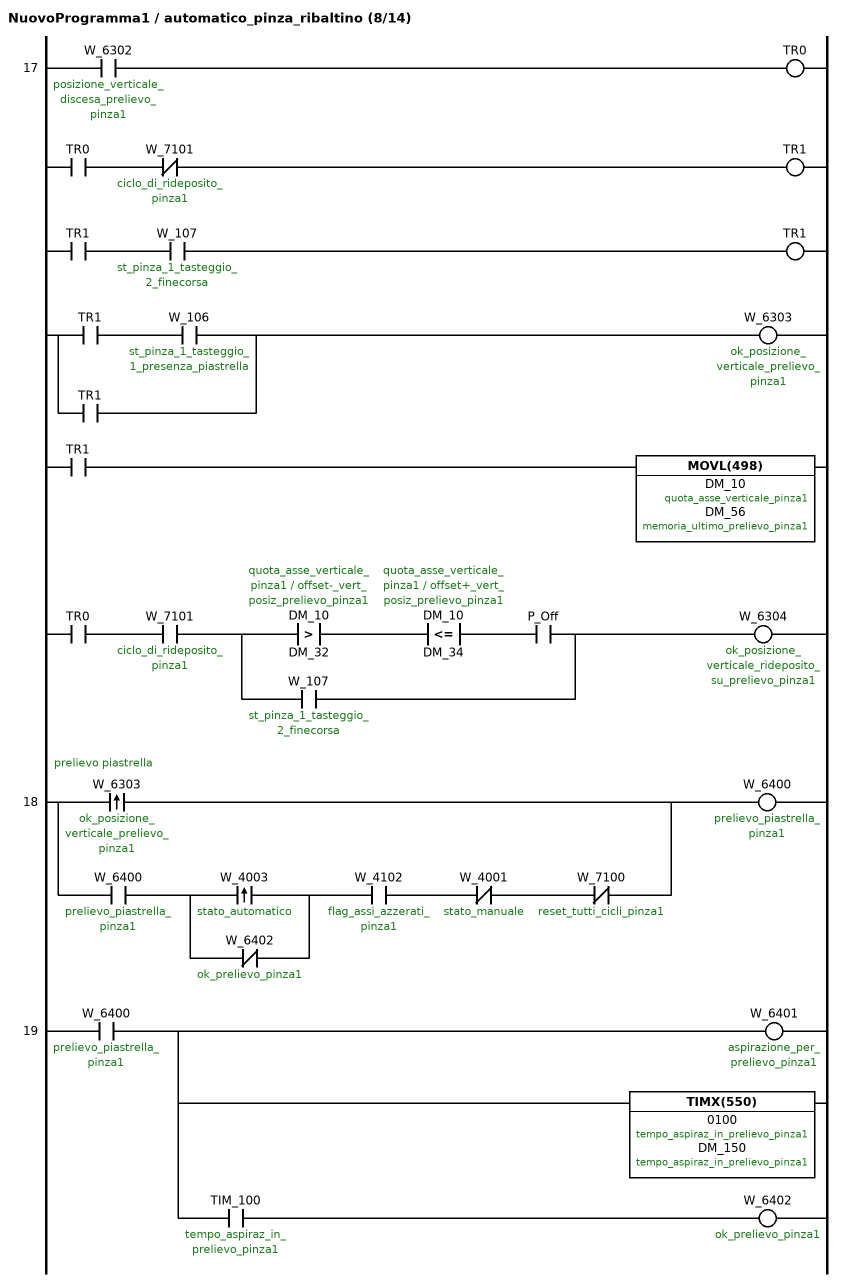
; [picture p48: NuovoProgramma1 / automatico_pinza_ribaltino, rungs 17-19]
; rung 17
LD W_6302  ; posizione_verticale_discesa_prelievo_pinza1
OUT TR0
ANDNOT W_7101  ; ciclo_di_rideposito_pinza1
OUT TR1
AND W_106  ; st_pinza_1_tasteggio_1_presenza_piastrella
LD TR1
AND W_107  ; st_pinza_1_tasteggio_2_finecorsa
OUT TR1
ORLD
OUT W_6303  ; ok_posizione_verticale_prelievo_pinza1
LD TR1
MOVL(498) DM_10 DM_56  ; quota_asse_verticale_pinza1, memoria_ultimo_prelievo_pinza1
LD TR0
AND W_7101  ; ciclo_di_rideposito_pinza1
LD>SL(323) DM_10 DM_32  ; quota_asse_verticale_pinza1, offset-_vert_posiz_prelievo_pinza1
AND<=SL(318) DM_10 DM_34  ; quota_asse_verticale_pinza1, offset+_vert_posiz_prelievo_pinza1
AND P_Off
OR W_107  ; st_pinza_1_tasteggio_2_finecorsa
ANDLD
OUT W_6304  ; ok_posizione_verticale_rideposito_su_prelievo_pinza1
; rung 18: prelievo piastrella
@LD W_6303  ; ok_posizione_verticale_prelievo_pinza1
LD W_6400  ; prelievo_piastrella_pinza1
@LD W_4003  ; stato_automatico
ORNOT W_6402  ; ok_prelievo_pinza1
ANDLD
AND W_4102  ; flag_assi_azzerati_pinza1
ANDNOT W_4001  ; stato_manuale
ANDNOT W_7100  ; reset_tutti_cicli_pinza1
ORLD
OUT W_6400  ; prelievo_piastrella_pinza1
; rung 19
LD W_6400  ; prelievo_piastrella_pinza1
OUT W_6401  ; aspirazione_per_prelievo_pinza1
TIMX(550) 0100 DM_150  ; tempo_aspiraz_in_prelievo_pinza1
AND TIM_100  ; tempo_aspiraz_in_prelievo_pinza1
OUT W_6402  ; ok_prelievo_pinza1

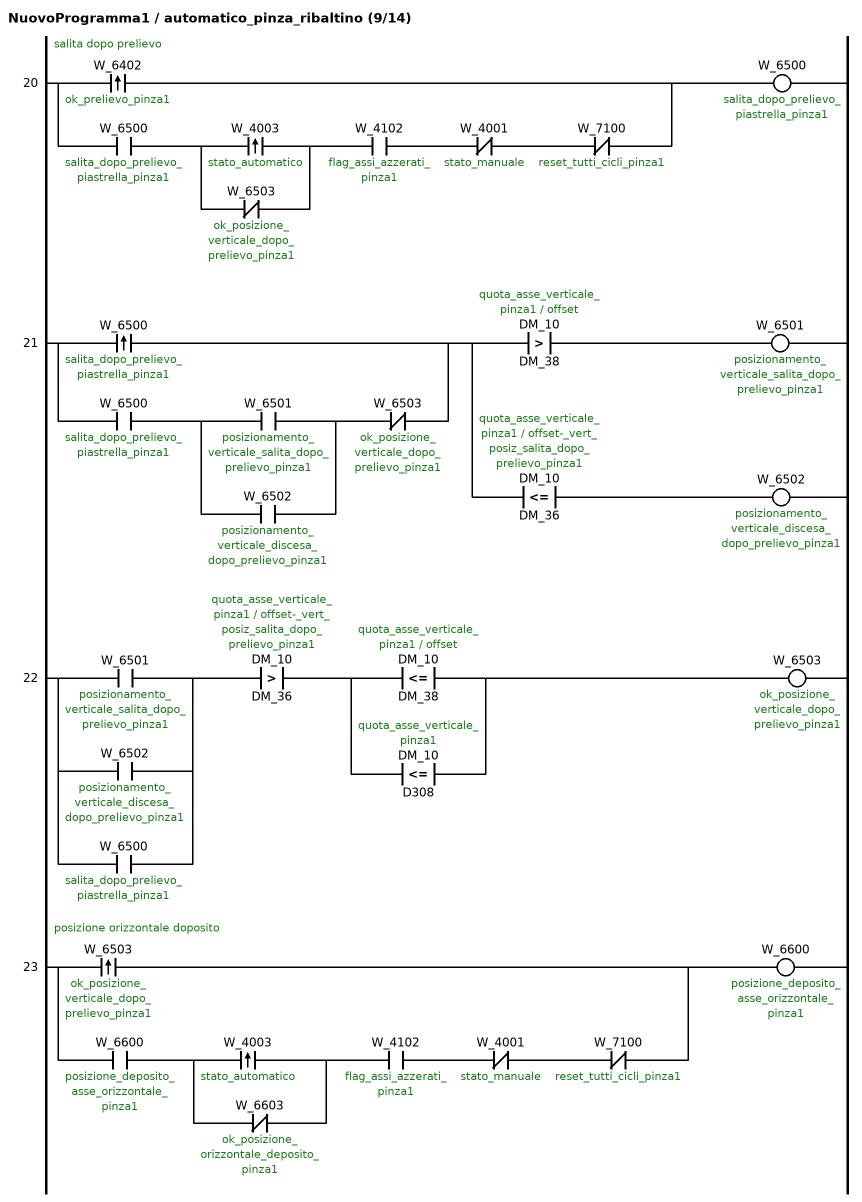
; rung 20: salita dopo prelievo
@LD W_6402  ; ok_prelievo_pinza1
LD W_6500  ; salita_dopo_prelievo_piastrella_pinza1
@LD W_4003  ; stato_automatico
ORNOT W_6503  ; ok_posizione_verticale_dopo_prelievo_pinza1
ANDLD
AND W_4102  ; flag_assi_azzerati_pinza1
ANDNOT W_4001  ; stato_manuale
ANDNOT W_7100  ; reset_tutti_cicli_pinza1
ORLD
OUT W_6500  ; salita_dopo_prelievo_piastrella_pinza1
; rung 21
@LD W_6500  ; salita_dopo_prelievo_piastrella_pinza1
LD W_6500  ; salita_dopo_prelievo_piastrella_pinza1
LD W_6501  ; posizionamento_verticale_salita_dopo_prelievo_pinza1
OR W_6502  ; posizionamento_verticale_discesa_dopo_prelievo_pinza1
ANDLD
ANDNOT W_6503  ; ok_posizione_verticale_dopo_prelievo_pinza1
ORLD
OUT TR0
AND>SL(323) DM_10 DM_38  ; quota_asse_verticale_pinza1, offset
OUT W_6501  ; posizionamento_verticale_salita_dopo_prelievo_pinza1
LD TR0
AND<=SL(318) DM_10 DM_36  ; quota_asse_verticale_pinza1, offset-_vert_posiz_salita_dopo_prelievo_pinza1
OUT W_6502  ; posizionamento_verticale_discesa_dopo_prelievo_pinza1
; rung 22
LD W_6501  ; posizionamento_verticale_salita_dopo_prelievo_pinza1
OR W_6502  ; posizionamento_verticale_discesa_dopo_prelievo_pinza1
OR W_6500  ; salita_dopo_prelievo_piastrella_pinza1
AND>SL(323) DM_10 DM_36  ; quota_asse_verticale_pinza1, offset-_vert_posiz_salita_dopo_prelievo_pinza1
LD<=SL(318) DM_10 DM_38  ; quota_asse_verticale_pinza1, offset
OR<=SL(318) DM_10 D308  ; quota_asse_verticale_pinza1
ANDLD
OUT W_6503  ; ok_posizione_verticale_dopo_prelievo_pinza1
; rung 23: posizione orizzontale doposito
@LD W_6503  ; ok_posizione_verticale_dopo_prelievo_pinza1
LD W_6600  ; posizione_deposito_asse_orizzontale_pinza1
@LD W_4003  ; stato_automatico
ORNOT W_6603  ; ok_posizione_orizzontale_deposito_pinza1
ANDLD
AND W_4102  ; flag_assi_azzerati_pinza1
ANDNOT W_4001  ; stato_manuale
ANDNOT W_7100  ; reset_tutti_cicli_pinza1
ORLD
OUT W_6600  ; posizione_deposito_asse_orizzontale_pinza1

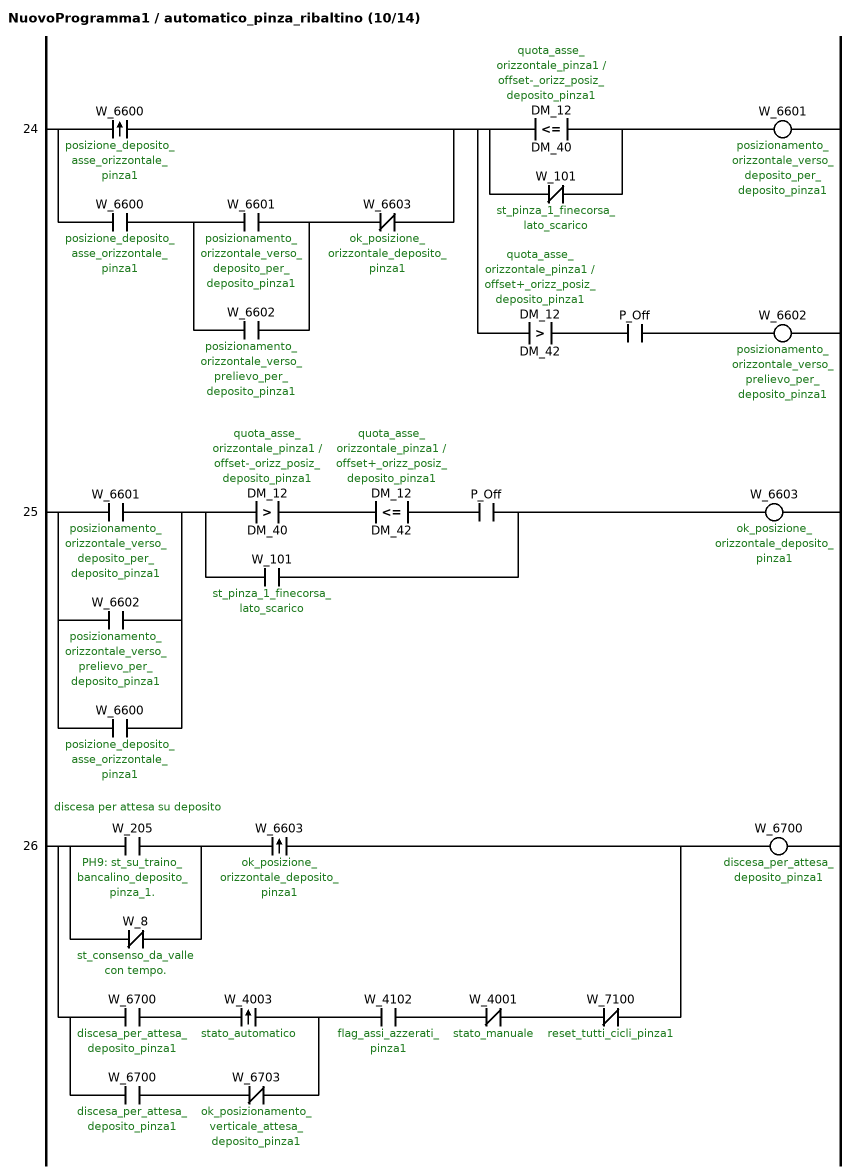
; rung 24
@LD W_6600  ; posizione_deposito_asse_orizzontale_pinza1
LD W_6600  ; posizione_deposito_asse_orizzontale_pinza1
LD W_6601  ; posizionamento_orizzontale_verso_deposito_per_deposito_pinza1
OR W_6602  ; posizionamento_orizzontale_verso_prelievo_per_deposito_pinza1
ANDLD
ANDNOT W_6603  ; ok_posizione_orizzontale_deposito_pinza1
ORLD
OUT TR0
LD<=SL(318) DM_12 DM_40  ; quota_asse_orizzontale_pinza1, offset-_orizz_posiz_deposito_pinza1
ORNOT W_101  ; st_pinza_1_finecorsa_lato_scarico
ANDLD
OUT W_6601  ; posizionamento_orizzontale_verso_deposito_per_deposito_pinza1
LD TR0
AND>SL(323) DM_12 DM_42  ; quota_asse_orizzontale_pinza1, offset+_orizz_posiz_deposito_pinza1
AND P_Off
OUT W_6602  ; posizionamento_orizzontale_verso_prelievo_per_deposito_pinza1
; rung 25
LD W_6601  ; posizionamento_orizzontale_verso_deposito_per_deposito_pinza1
OR W_6602  ; posizionamento_orizzontale_verso_prelievo_per_deposito_pinza1
OR W_6600  ; posizione_deposito_asse_orizzontale_pinza1
LD>SL(323) DM_12 DM_40  ; quota_asse_orizzontale_pinza1, offset-_orizz_posiz_deposito_pinza1
AND<=SL(318) DM_12 DM_42  ; quota_asse_orizzontale_pinza1, offset+_orizz_posiz_deposito_pinza1
AND P_Off
OR W_101  ; st_pinza_1_finecorsa_lato_scarico
ANDLD
OUT W_6603  ; ok_posizione_orizzontale_deposito_pinza1
; rung 26: discesa per attesa su deposito
LD W_205  ; PH9: st_su_traino_bancalino_deposito_pinza_1.
ORNOT W_8  ; st_consenso_da_valle con tempo.
@AND W_6603  ; ok_posizione_orizzontale_deposito_pinza1
LD W_6700  ; discesa_per_attesa_deposito_pinza1
@AND W_4003  ; stato_automatico
LD W_6700  ; discesa_per_attesa_deposito_pinza1
ANDNOT W_6703  ; ok_posizionamento_verticale_attesa_deposito_pinza1
ORLD
AND W_4102  ; flag_assi_azzerati_pinza1
ANDNOT W_4001  ; stato_manuale
ANDNOT W_7100  ; reset_tutti_cicli_pinza1
ORLD
OUT W_6700  ; discesa_per_attesa_deposito_pinza1

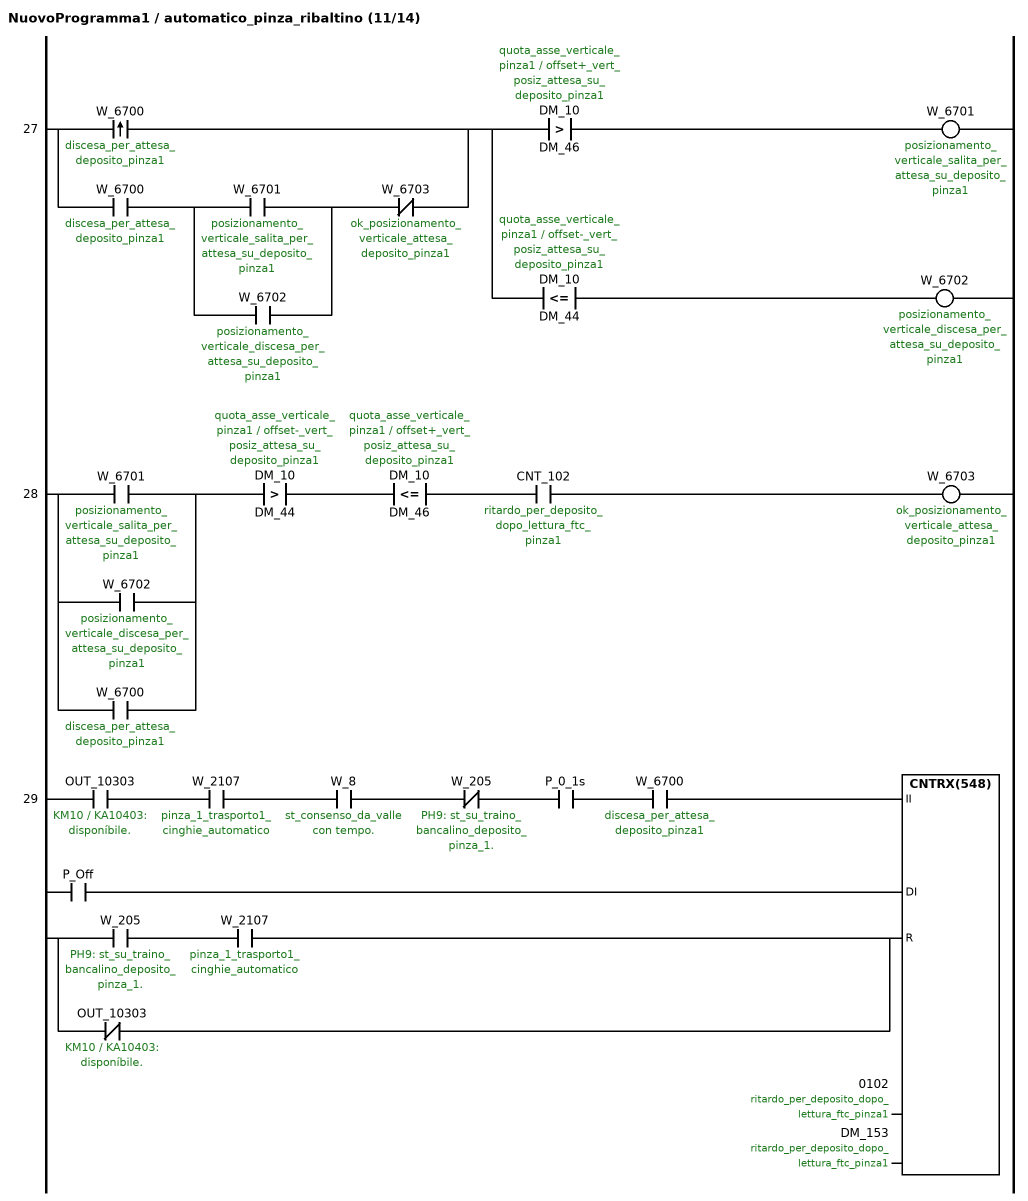
; rung 27
@LD W_6700  ; discesa_per_attesa_deposito_pinza1
LD W_6700  ; discesa_per_attesa_deposito_pinza1
LD W_6701  ; posizionamento_verticale_salita_per_attesa_su_deposito_pinza1
OR W_6702  ; posizionamento_verticale_discesa_per_attesa_su_deposito_pinza1
ANDLD
ANDNOT W_6703  ; ok_posizionamento_verticale_attesa_deposito_pinza1
ORLD
OUT TR0
AND>SL(323) DM_10 DM_46  ; quota_asse_verticale_pinza1, offset+_vert_posiz_attesa_su_deposito_pinza1
OUT W_6701  ; posizionamento_verticale_salita_per_attesa_su_deposito_pinza1
LD TR0
AND<=SL(318) DM_10 DM_44  ; quota_asse_verticale_pinza1, offset-_vert_posiz_attesa_su_deposito_pinza1
OUT W_6702  ; posizionamento_verticale_discesa_per_attesa_su_deposito_pinza1
; rung 28
LD W_6701  ; posizionamento_verticale_salita_per_attesa_su_deposito_pinza1
OR W_6702  ; posizionamento_verticale_discesa_per_attesa_su_deposito_pinza1
OR W_6700  ; discesa_per_attesa_deposito_pinza1
AND>SL(323) DM_10 DM_44  ; quota_asse_verticale_pinza1, offset-_vert_posiz_attesa_su_deposito_pinza1
AND<=SL(318) DM_10 DM_46  ; quota_asse_verticale_pinza1, offset+_vert_posiz_attesa_su_deposito_pinza1
AND CNT_102  ; ritardo_per_deposito_dopo_lettura_ftc_pinza1
OUT W_6703  ; ok_posizionamento_verticale_attesa_deposito_pinza1
; rung 29
LD OUT_10303  ; KM10 / KA10403: disponíbile.
AND W_2107  ; pinza_1_trasporto1_cinghie_automatico
AND W_8  ; st_consenso_da_valle con tempo.
ANDNOT W_205  ; PH9: st_su_traino_bancalino_deposito_pinza_1.
AND P_0_1s
AND W_6700  ; discesa_per_attesa_deposito_pinza1
LD P_Off
LD W_205  ; PH9: st_su_traino_bancalino_deposito_pinza_1.
AND W_2107  ; pinza_1_trasporto1_cinghie_automatico
ORNOT OUT_10303  ; KM10 / KA10403: disponíbile.
CNTRX(548) 0102 DM_153  ; ritardo_per_deposito_dopo_lettura_ftc_pinza1

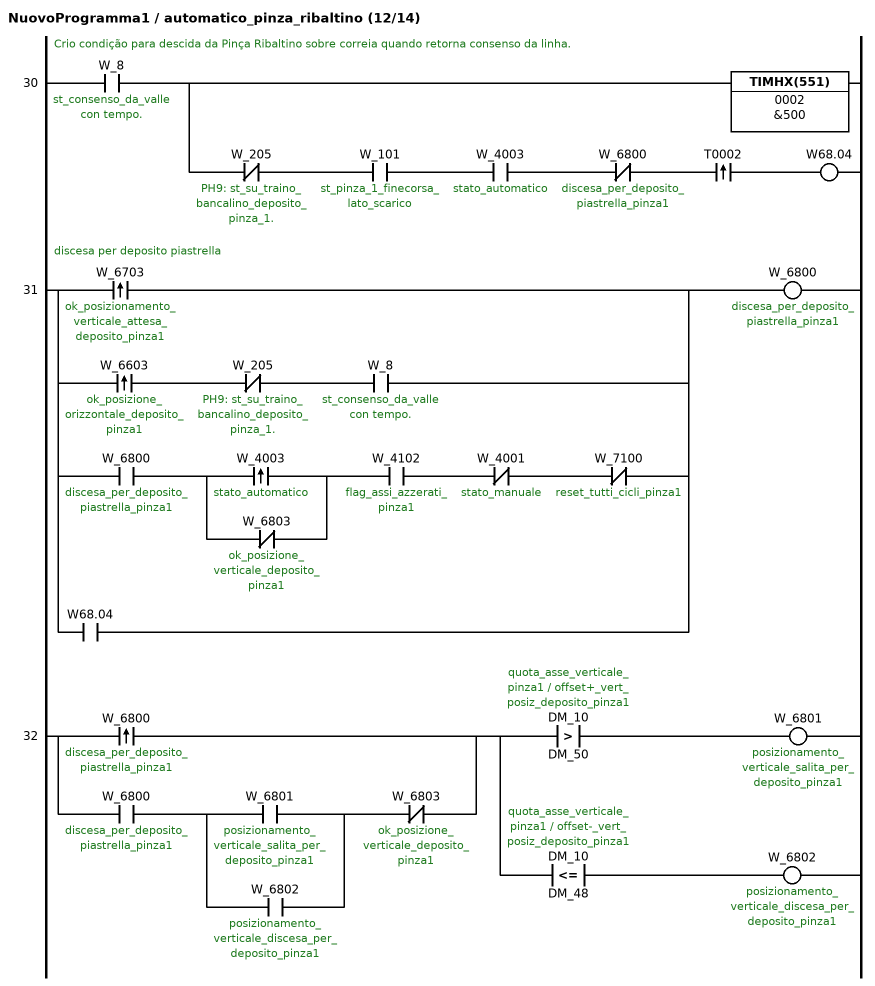
; rung 30: Crio condição para descida da Pinça Ribaltino sobre correia quando retorna consenso da linha.
LD W_8  ; st_consenso_da_valle con tempo.
TIMHX(551) 0002 &500
ANDNOT W_205  ; PH9: st_su_traino_bancalino_deposito_pinza_1.
AND W_101  ; st_pinza_1_finecorsa_lato_scarico
AND W_4003  ; stato_automatico
ANDNOT W_6800  ; discesa_per_deposito_piastrella_pinza1
@AND T0002
OUT W68.04
; rung 31: discesa per deposito piastrella
@LD W_6703  ; ok_posizionamento_verticale_attesa_deposito_pinza1
@LD W_6603  ; ok_posizione_orizzontale_deposito_pinza1
ANDNOT W_205  ; PH9: st_su_traino_bancalino_deposito_pinza_1.
AND W_8  ; st_consenso_da_valle con tempo.
ORLD
LD W_6800  ; discesa_per_deposito_piastrella_pinza1
@LD W_4003  ; stato_automatico
ORNOT W_6803  ; ok_posizione_verticale_deposito_pinza1
ANDLD
AND W_4102  ; flag_assi_azzerati_pinza1
ANDNOT W_4001  ; stato_manuale
ANDNOT W_7100  ; reset_tutti_cicli_pinza1
ORLD
OR W68.04
OUT W_6800  ; discesa_per_deposito_piastrella_pinza1
; rung 32
@LD W_6800  ; discesa_per_deposito_piastrella_pinza1
LD W_6800  ; discesa_per_deposito_piastrella_pinza1
LD W_6801  ; posizionamento_verticale_salita_per_deposito_pinza1
OR W_6802  ; posizionamento_verticale_discesa_per_deposito_pinza1
ANDLD
ANDNOT W_6803  ; ok_posizione_verticale_deposito_pinza1
ORLD
OUT TR0
AND>SL(323) DM_10 DM_50  ; quota_asse_verticale_pinza1, offset+_vert_posiz_deposito_pinza1
OUT W_6801  ; posizionamento_verticale_salita_per_deposito_pinza1
LD TR0
AND<=SL(318) DM_10 DM_48  ; quota_asse_verticale_pinza1, offset-_vert_posiz_deposito_pinza1
OUT W_6802  ; posizionamento_verticale_discesa_per_deposito_pinza1

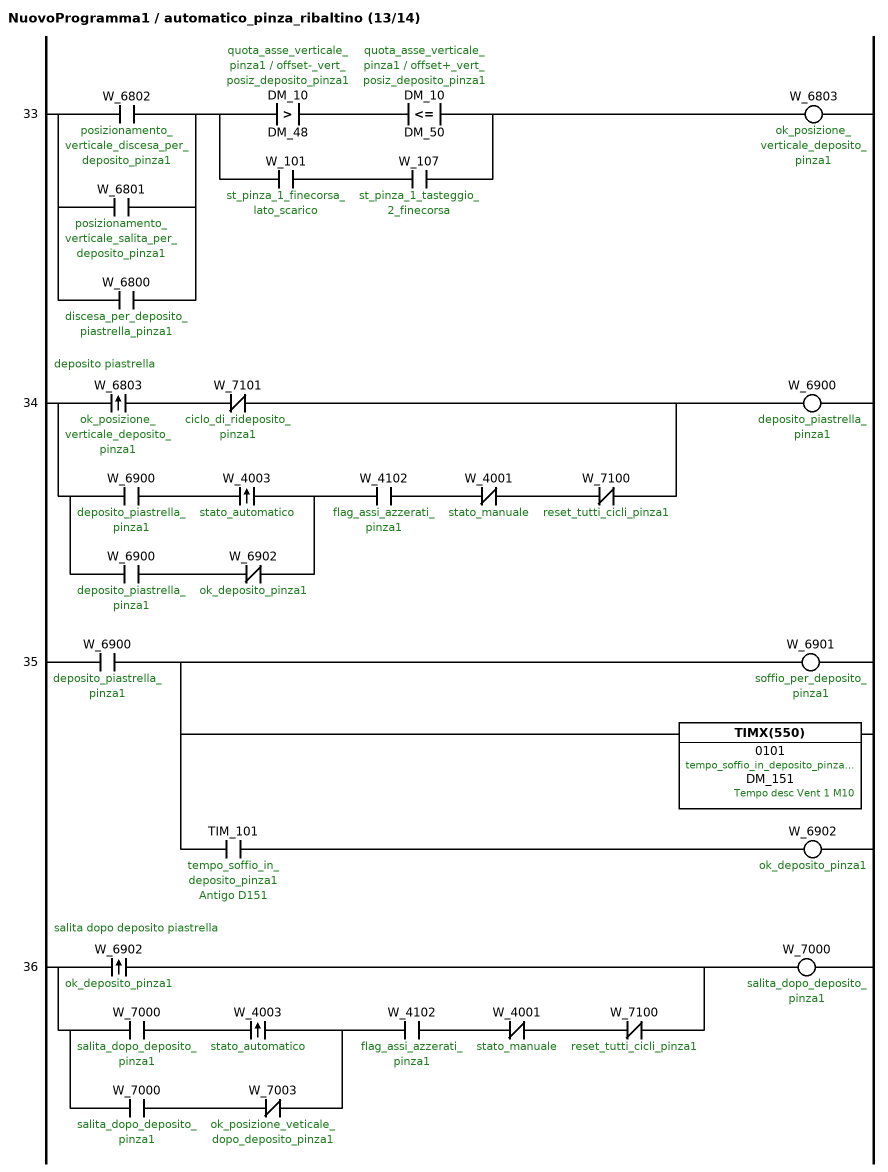
; rung 33
LD W_6802  ; posizionamento_verticale_discesa_per_deposito_pinza1
OR W_6801  ; posizionamento_verticale_salita_per_deposito_pinza1
OR W_6800  ; discesa_per_deposito_piastrella_pinza1
LD>SL(323) DM_10 DM_48  ; quota_asse_verticale_pinza1, offset-_vert_posiz_deposito_pinza1
AND<=SL(318) DM_10 DM_50  ; quota_asse_verticale_pinza1, offset+_vert_posiz_deposito_pinza1
LD W_101  ; st_pinza_1_finecorsa_lato_scarico
AND W_107  ; st_pinza_1_tasteggio_2_finecorsa
ORLD
ANDLD
OUT W_6803  ; ok_posizione_verticale_deposito_pinza1
; rung 34: deposito piastrella
@LD W_6803  ; ok_posizione_verticale_deposito_pinza1
ANDNOT W_7101  ; ciclo_di_rideposito_pinza1
LD W_6900  ; deposito_piastrella_pinza1
@AND W_4003  ; stato_automatico
LD W_6900  ; deposito_piastrella_pinza1
ANDNOT W_6902  ; ok_deposito_pinza1
ORLD
AND W_4102  ; flag_assi_azzerati_pinza1
ANDNOT W_4001  ; stato_manuale
ANDNOT W_7100  ; reset_tutti_cicli_pinza1
ORLD
OUT W_6900  ; deposito_piastrella_pinza1
; rung 35
LD W_6900  ; deposito_piastrella_pinza1
OUT W_6901  ; soffio_per_deposito_pinza1
TIMX(550) 0101 DM_151  ; Tempo desc Vent 1 M10, tempo_soffio_in_deposito_pinza1 Antigo D151
AND TIM_101  ; tempo_soffio_in_deposito_pinza1 Antigo D151
OUT W_6902  ; ok_deposito_pinza1
; rung 36: salita dopo deposito piastrella
@LD W_6902  ; ok_deposito_pinza1
LD W_7000  ; salita_dopo_deposito_pinza1
@AND W_4003  ; stato_automatico
LD W_7000  ; salita_dopo_deposito_pinza1
ANDNOT W_7003  ; ok_posizione_veticale_dopo_deposito_pinza1
ORLD
AND W_4102  ; flag_assi_azzerati_pinza1
ANDNOT W_4001  ; stato_manuale
ANDNOT W_7100  ; reset_tutti_cicli_pinza1
ORLD
OUT W_7000  ; salita_dopo_deposito_pinza1

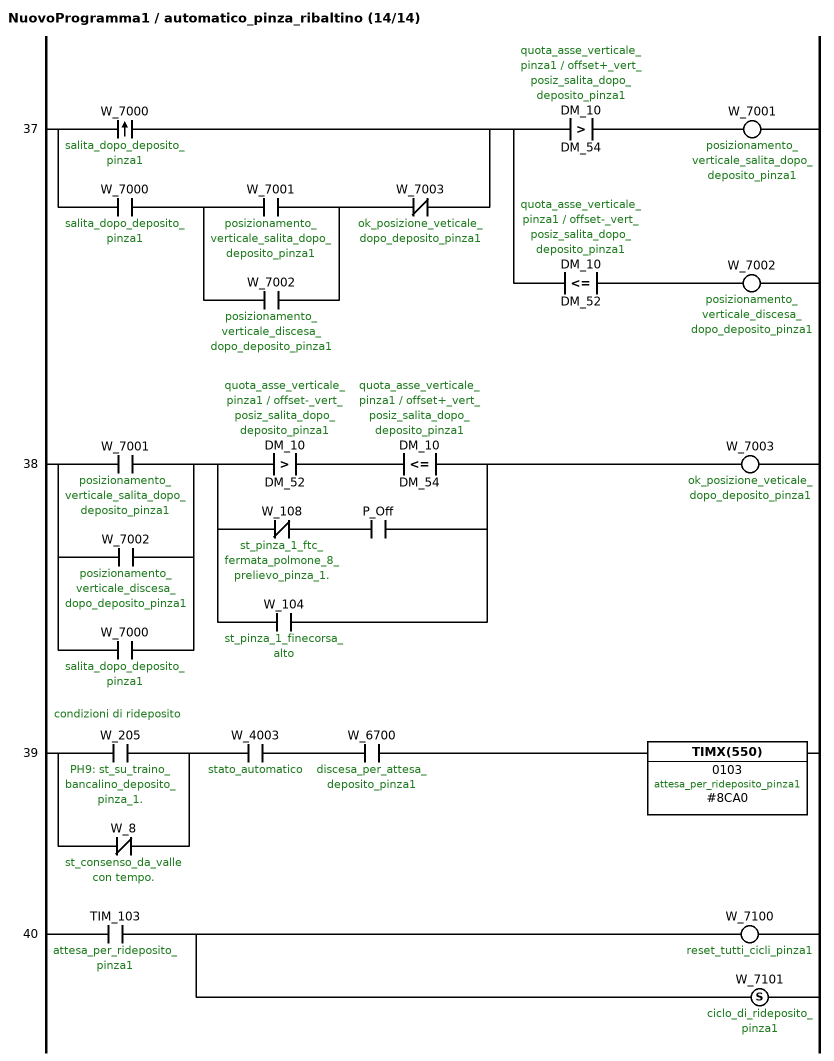
; rung 37
@LD W_7000  ; salita_dopo_deposito_pinza1
LD W_7000  ; salita_dopo_deposito_pinza1
LD W_7001  ; posizionamento_verticale_salita_dopo_deposito_pinza1
OR W_7002  ; posizionamento_verticale_discesa_dopo_deposito_pinza1
ANDLD
ANDNOT W_7003  ; ok_posizione_veticale_dopo_deposito_pinza1
ORLD
OUT TR0
AND>SL(323) DM_10 DM_54  ; quota_asse_verticale_pinza1, offset+_vert_posiz_salita_dopo_deposito_pinza1
OUT W_7001  ; posizionamento_verticale_salita_dopo_deposito_pinza1
LD TR0
AND<=SL(318) DM_10 DM_52  ; quota_asse_verticale_pinza1, offset-_vert_posiz_salita_dopo_deposito_pinza1
OUT W_7002  ; posizionamento_verticale_discesa_dopo_deposito_pinza1
; rung 38
LD W_7001  ; posizionamento_verticale_salita_dopo_deposito_pinza1
OR W_7002  ; posizionamento_verticale_discesa_dopo_deposito_pinza1
OR W_7000  ; salita_dopo_deposito_pinza1
LD>SL(323) DM_10 DM_52  ; quota_asse_verticale_pinza1, offset-_vert_posiz_salita_dopo_deposito_pinza1
AND<=SL(318) DM_10 DM_54  ; quota_asse_verticale_pinza1, offset+_vert_posiz_salita_dopo_deposito_pinza1
LDNOT W_108  ; st_pinza_1_ftc_fermata_polmone_8_prelievo_pinza_1.
AND P_Off
ORLD
OR W_104  ; st_pinza_1_finecorsa_alto
ANDLD
OUT W_7003  ; ok_posizione_veticale_dopo_deposito_pinza1
; rung 39: condizioni di rideposito
LD W_205  ; PH9: st_su_traino_bancalino_deposito_pinza_1.
ORNOT W_8  ; st_consenso_da_valle con tempo.
AND W_4003  ; stato_automatico
AND W_6700  ; discesa_per_attesa_deposito_pinza1
TIMX(550) 0103 #8CA0  ; attesa_per_rideposito_pinza1
; rung 40
LD TIM_103  ; attesa_per_rideposito_pinza1
OUT W_7100  ; reset_tutti_cicli_pinza1
SET W_7101  ; ciclo_di_rideposito_pinza1

### Section rulliera_carico_ribaltino

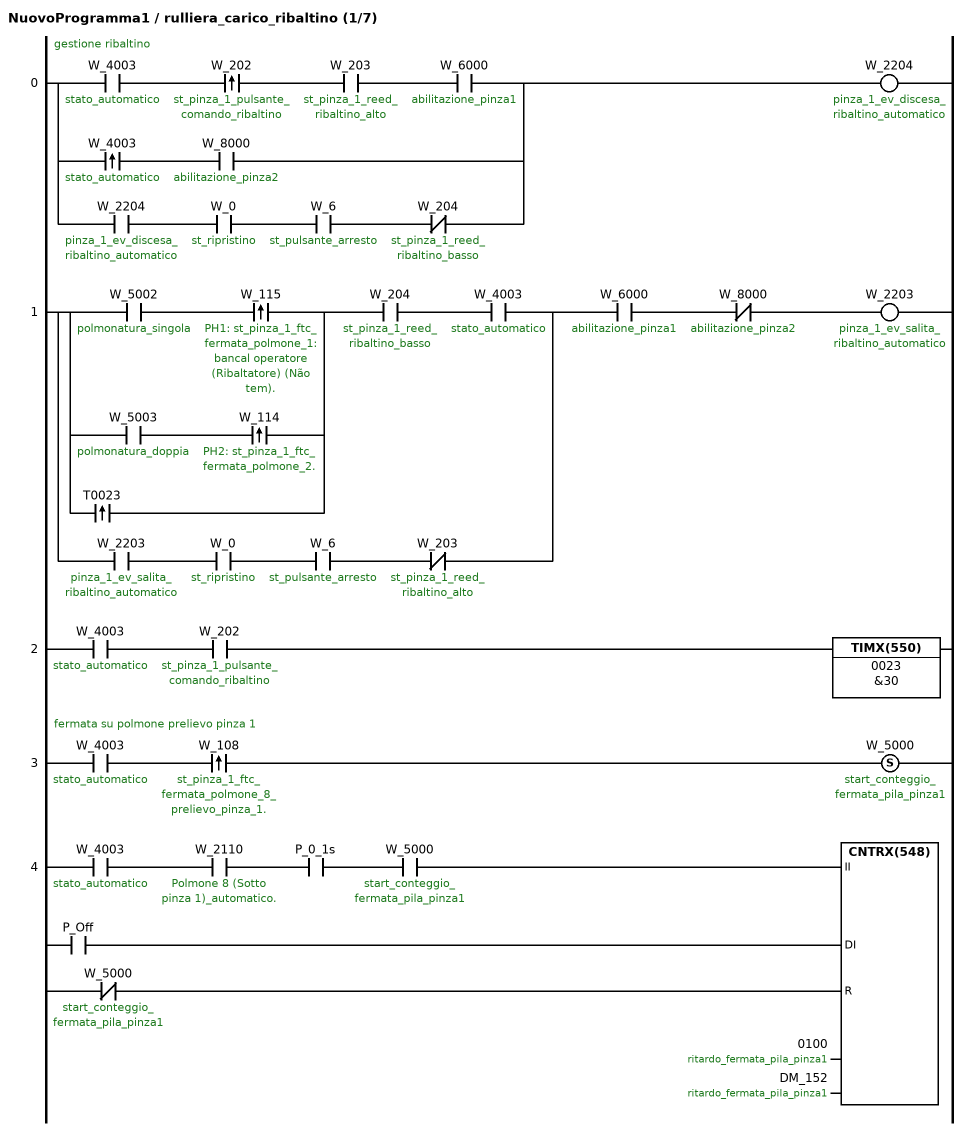
; rung 0: gestione ribaltino
LD W_4003  ; stato_automatico
@AND W_202  ; st_pinza_1_pulsante_comando_ribaltino
AND W_203  ; st_pinza_1_reed_ribaltino_alto
AND W_6000  ; abilitazione_pinza1
@LD W_4003  ; stato_automatico
AND W_8000  ; abilitazione_pinza2
ORLD
LD W_2204  ; pinza_1_ev_discesa_ribaltino_automatico
AND W_0  ; st_ripristino
AND W_6  ; st_pulsante_arresto
ANDNOT W_204  ; st_pinza_1_reed_ribaltino_basso
ORLD
OUT W_2204  ; pinza_1_ev_discesa_ribaltino_automatico
; rung 1
LD W_5002  ; polmonatura_singola
@AND W_115  ; PH1: st_pinza_1_ftc_fermata_polmone_1: bancal operatore (Ribaltatore) (Não tem).
LD W_5003  ; polmonatura_doppia
@AND W_114  ; PH2: st_pinza_1_ftc_fermata_polmone_2.
ORLD
@OR T0023
AND W_204  ; st_pinza_1_reed_ribaltino_basso
AND W_4003  ; stato_automatico
LD W_2203  ; pinza_1_ev_salita_ribaltino_automatico
AND W_0  ; st_ripristino
AND W_6  ; st_pulsante_arresto
ANDNOT W_203  ; st_pinza_1_reed_ribaltino_alto
ORLD
AND W_6000  ; abilitazione_pinza1
ANDNOT W_8000  ; abilitazione_pinza2
OUT W_2203  ; pinza_1_ev_salita_ribaltino_automatico
; rung 2
LD W_4003  ; stato_automatico
AND W_202  ; st_pinza_1_pulsante_comando_ribaltino
TIMX(550) 0023 &30
; rung 3: fermata su polmone prelievo pinza 1
LD W_4003  ; stato_automatico
@AND W_108  ; st_pinza_1_ftc_fermata_polmone_8_prelievo_pinza_1.
SET W_5000  ; start_conteggio_fermata_pila_pinza1
; rung 4
LD W_4003  ; stato_automatico
AND W_2110  ; Polmone 8 (Sotto pinza 1)_automatico.
AND P_0_1s
AND W_5000  ; start_conteggio_fermata_pila_pinza1
LD P_Off
LDNOT W_5000  ; start_conteggio_fermata_pila_pinza1
CNTRX(548) 0100 DM_152  ; ritardo_fermata_pila_pinza1

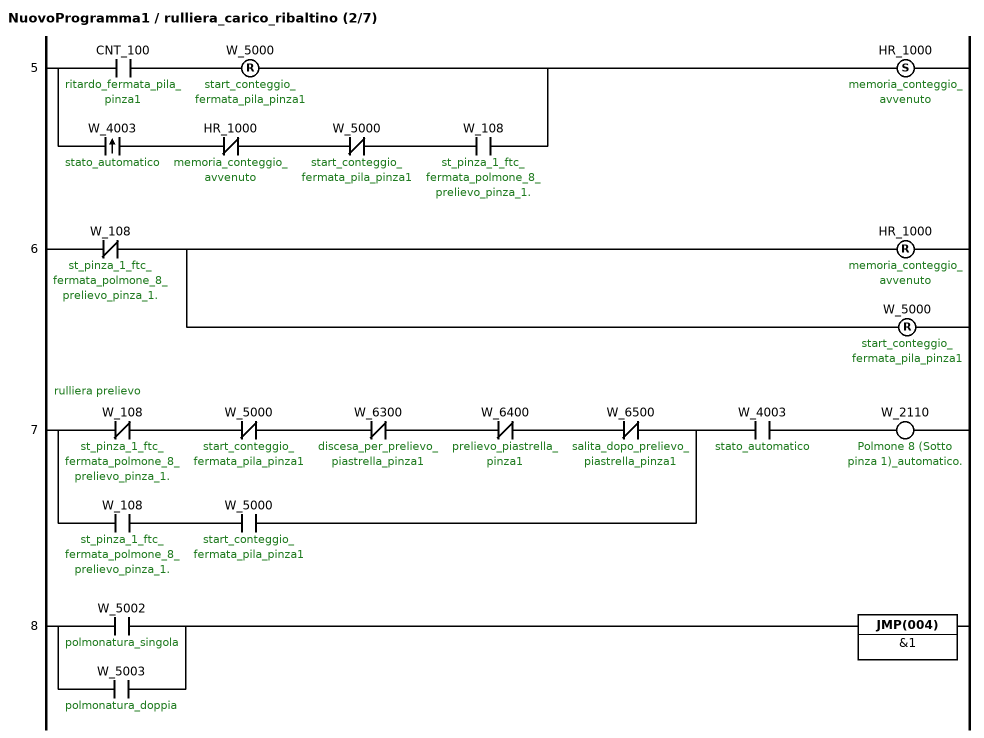
; rung 5
LD CNT_100  ; ritardo_fermata_pila_pinza1
RSET W_5000  ; start_conteggio_fermata_pila_pinza1
@LD W_4003  ; stato_automatico
ANDNOT HR_1000  ; memoria_conteggio_avvenuto
ANDNOT W_5000  ; start_conteggio_fermata_pila_pinza1
AND W_108  ; st_pinza_1_ftc_fermata_polmone_8_prelievo_pinza_1.
ORLD
SET HR_1000  ; memoria_conteggio_avvenuto
; rung 6
LDNOT W_108  ; st_pinza_1_ftc_fermata_polmone_8_prelievo_pinza_1.
RSET HR_1000  ; memoria_conteggio_avvenuto
RSET W_5000  ; start_conteggio_fermata_pila_pinza1
; rung 7: rulliera prelievo
LDNOT W_108  ; st_pinza_1_ftc_fermata_polmone_8_prelievo_pinza_1.
ANDNOT W_5000  ; start_conteggio_fermata_pila_pinza1
ANDNOT W_6300  ; discesa_per_prelievo_piastrella_pinza1
ANDNOT W_6400  ; prelievo_piastrella_pinza1
ANDNOT W_6500  ; salita_dopo_prelievo_piastrella_pinza1
LD W_108  ; st_pinza_1_ftc_fermata_polmone_8_prelievo_pinza_1.
AND W_5000  ; start_conteggio_fermata_pila_pinza1
ORLD
AND W_4003  ; stato_automatico
OUT W_2110  ; Polmone 8 (Sotto pinza 1)_automatico.
; rung 8
LD W_5002  ; polmonatura_singola
OR W_5003  ; polmonatura_doppia
JMP(004) &1

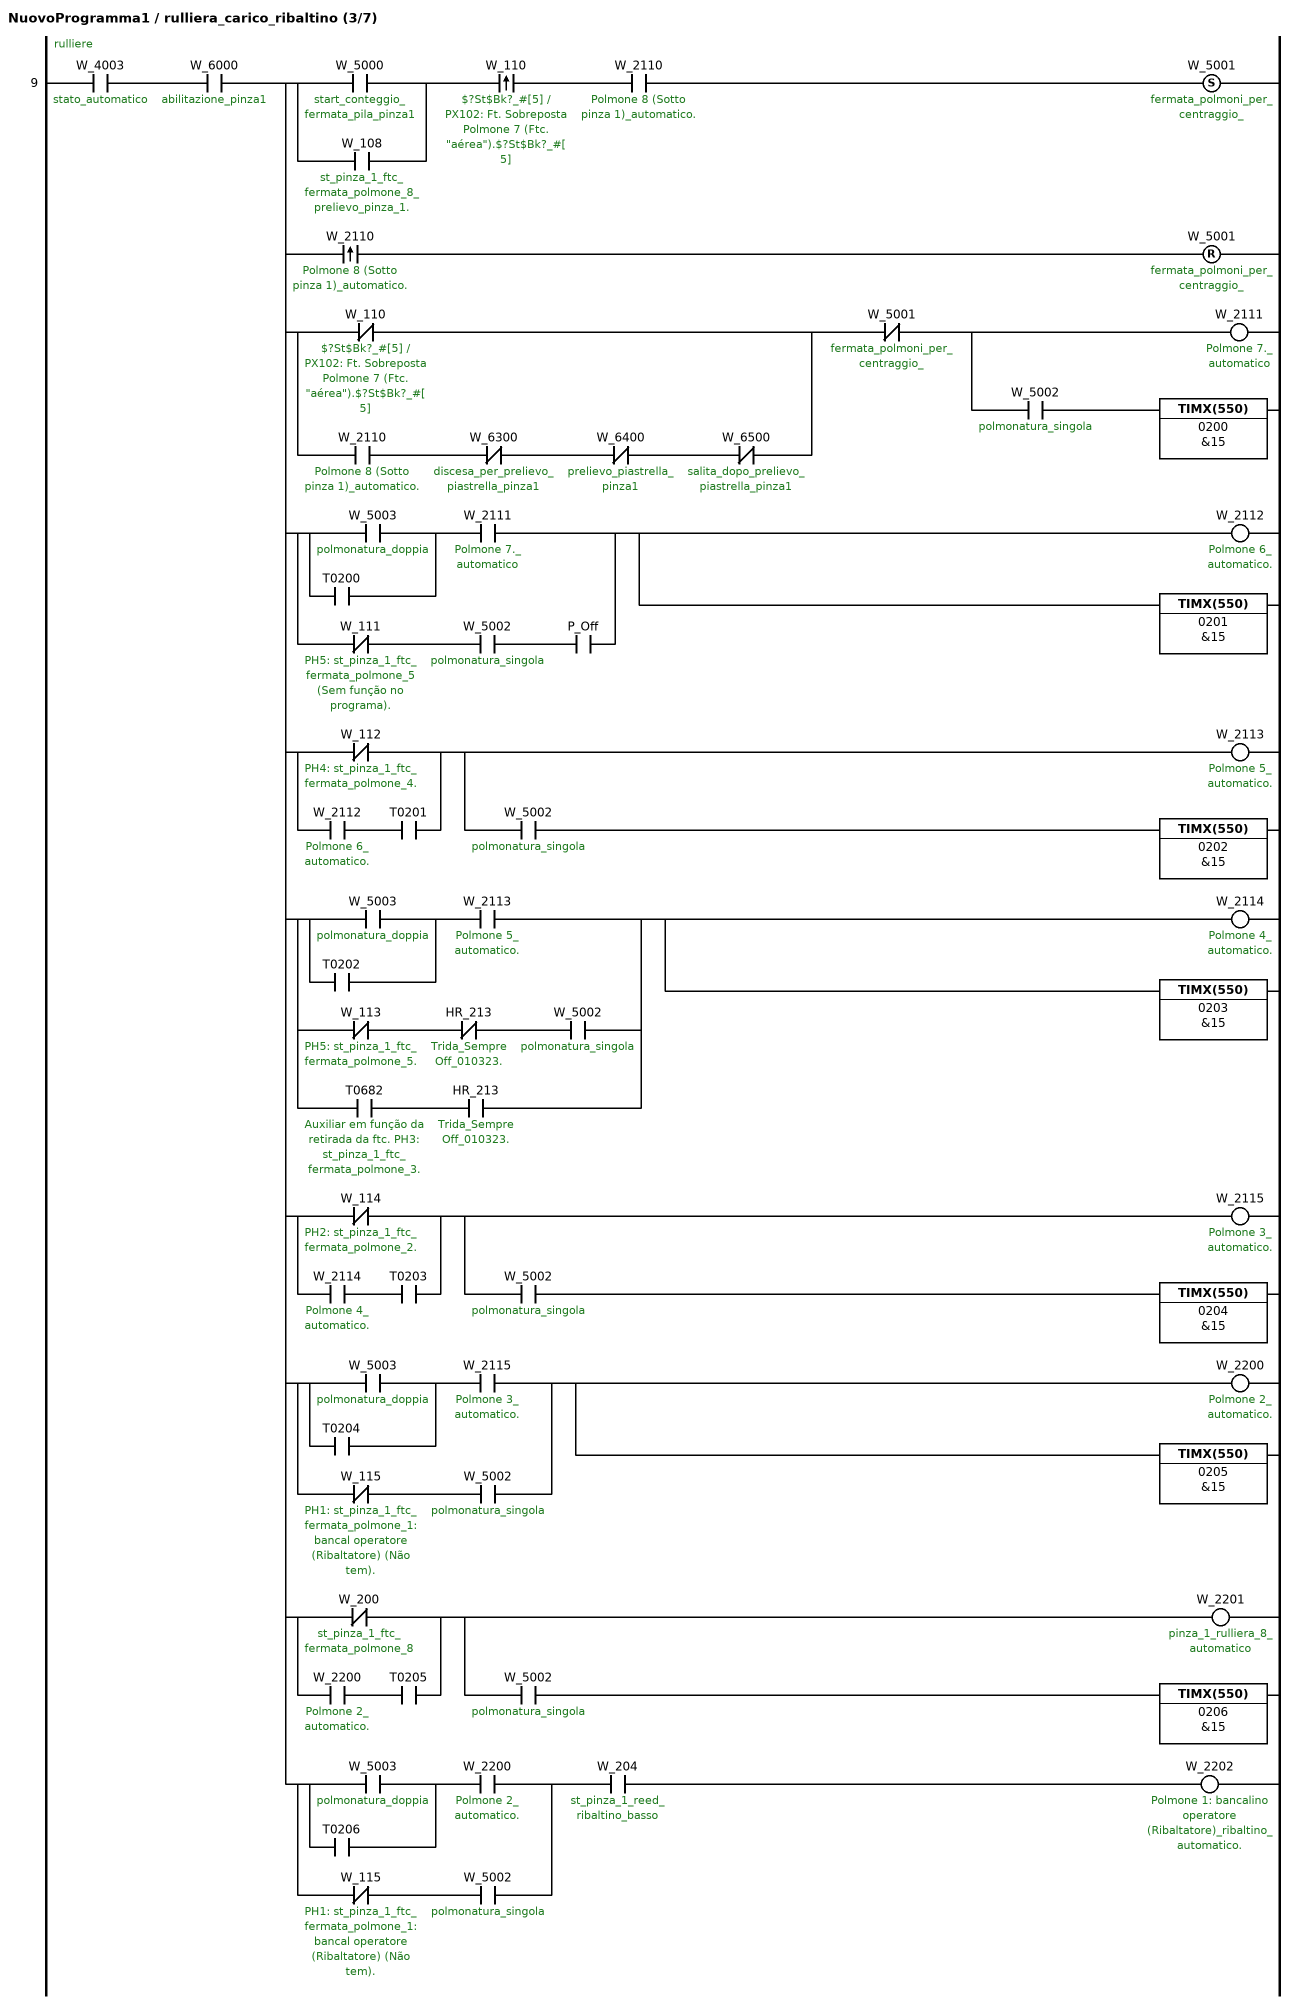
; rung 9: rulliere
LD W_4003  ; stato_automatico
AND W_6000  ; abilitazione_pinza1
OUT TR0
LD W_5000  ; start_conteggio_fermata_pila_pinza1
OR W_108  ; st_pinza_1_ftc_fermata_polmone_8_prelievo_pinza_1.
ANDLD
@AND W_110  ; $?St$Bk?_#[5] / PX102: Ft. Sobreposta Polmone 7 (Ftc. "aérea").$?St$Bk?_#[5]
AND W_2110  ; Polmone 8 (Sotto pinza 1)_automatico.
SET W_5001  ; fermata_polmoni_per_centraggio_
LD TR0
@AND W_2110  ; Polmone 8 (Sotto pinza 1)_automatico.
RSET W_5001  ; fermata_polmoni_per_centraggio_
LD TR0
LDNOT W_110  ; $?St$Bk?_#[5] / PX102: Ft. Sobreposta Polmone 7 (Ftc. "aérea").$?St$Bk?_#[5]
LD W_2110  ; Polmone 8 (Sotto pinza 1)_automatico.
ANDNOT W_6300  ; discesa_per_prelievo_piastrella_pinza1
ANDNOT W_6400  ; prelievo_piastrella_pinza1
ANDNOT W_6500  ; salita_dopo_prelievo_piastrella_pinza1
ORLD
ANDLD
ANDNOT W_5001  ; fermata_polmoni_per_centraggio_
OUT W_2111  ; Polmone 7._automatico
AND W_5002  ; polmonatura_singola
TIMX(550) 0200 &15
LD TR0
LD W_5003  ; polmonatura_doppia
OR T0200
AND W_2111  ; Polmone 7._automatico
LDNOT W_111  ; PH5: st_pinza_1_ftc_fermata_polmone_5 (Sem função no programa).
AND W_5002  ; polmonatura_singola
AND P_Off
ORLD
ANDLD
OUT W_2112  ; Polmone 6_automatico.
TIMX(550) 0201 &15
LD TR0
LDNOT W_112  ; PH4: st_pinza_1_ftc_fermata_polmone_4.
LD W_2112  ; Polmone 6_automatico.
AND T0201
ORLD
ANDLD
OUT W_2113  ; Polmone 5_automatico.
AND W_5002  ; polmonatura_singola
TIMX(550) 0202 &15
LD TR0
LD W_5003  ; polmonatura_doppia
OR T0202
AND W_2113  ; Polmone 5_automatico.
LDNOT W_113  ; PH5: st_pinza_1_ftc_fermata_polmone_5.
ANDNOT HR_213  ; Trida_Sempre Off_010323.
AND W_5002  ; polmonatura_singola
ORLD
LD T0682  ; Auxiliar em função da retirada da ftc. PH3: st_pinza_1_ftc_fermata_polmone_3.
AND HR_213  ; Trida_Sempre Off_010323.
ORLD
ANDLD
OUT W_2114  ; Polmone 4_automatico.
TIMX(550) 0203 &15
LD TR0
LDNOT W_114  ; PH2: st_pinza_1_ftc_fermata_polmone_2.
LD W_2114  ; Polmone 4_automatico.
AND T0203
ORLD
ANDLD
OUT W_2115  ; Polmone 3_automatico.
AND W_5002  ; polmonatura_singola
TIMX(550) 0204 &15
LD TR0
LD W_5003  ; polmonatura_doppia
OR T0204
AND W_2115  ; Polmone 3_automatico.
LDNOT W_115  ; PH1: st_pinza_1_ftc_fermata_polmone_1: bancal operatore (Ribaltatore) (Não tem).
AND W_5002  ; polmonatura_singola
ORLD
ANDLD
OUT W_2200  ; Polmone 2_automatico.
TIMX(550) 0205 &15
LD TR0
LDNOT W_200  ; st_pinza_1_ftc_fermata_polmone_8
LD W_2200  ; Polmone 2_automatico.
AND T0205
ORLD
ANDLD
OUT W_2201  ; pinza_1_rulliera_8_automatico
AND W_5002  ; polmonatura_singola
TIMX(550) 0206 &15
LD TR0
LD W_5003  ; polmonatura_doppia
OR T0206
AND W_2200  ; Polmone 2_automatico.
LDNOT W_115  ; PH1: st_pinza_1_ftc_fermata_polmone_1: bancal operatore (Ribaltatore) (Não tem).
AND W_5002  ; polmonatura_singola
ORLD
ANDLD
AND W_204  ; st_pinza_1_reed_ribaltino_basso
OUT W_2202  ; Polmone 1: bancalino operatore (Ribaltatore)_ribaltino_automatico.

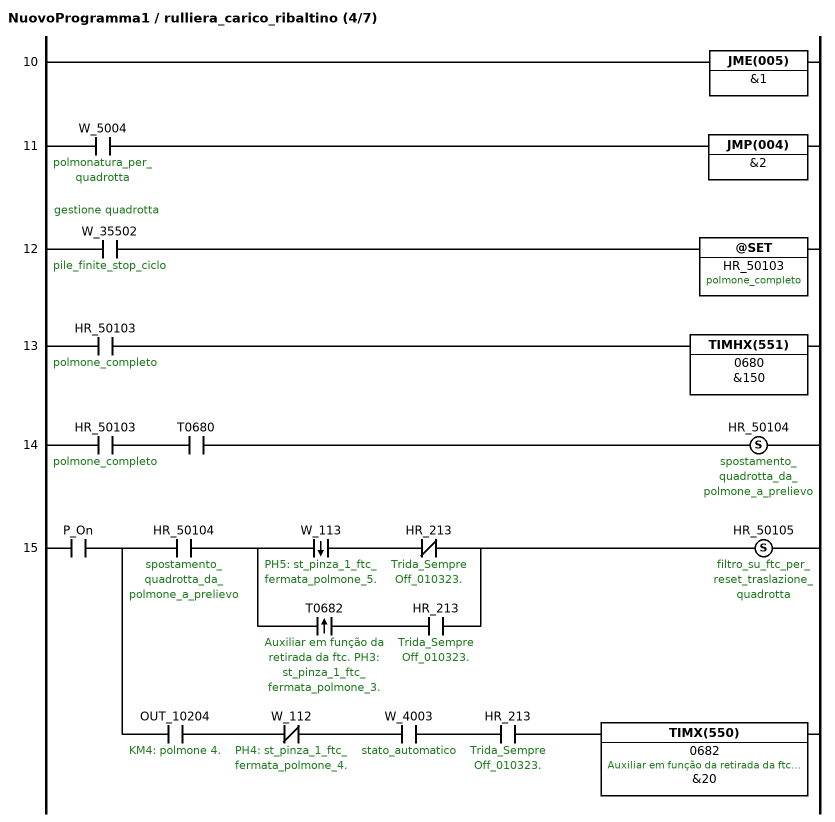
; rung 10
JME(005) &1
; rung 11
LD W_5004  ; polmonatura_per_quadrotta
JMP(004) &2
; rung 12: gestione quadrotta
LD W_35502  ; pile_finite_stop_ciclo
@SET HR_50103  ; polmone_completo
; rung 13
LD HR_50103  ; polmone_completo
TIMHX(551) 0680 &150
; rung 14
LD HR_50103  ; polmone_completo
AND T0680
SET HR_50104  ; spostamento_quadrotta_da_polmone_a_prelievo
; rung 15
LD P_On
OUT TR0
AND HR_50104  ; spostamento_quadrotta_da_polmone_a_prelievo
%LD W_113  ; PH5: st_pinza_1_ftc_fermata_polmone_5.
ANDNOT HR_213  ; Trida_Sempre Off_010323.
@LD T0682  ; Auxiliar em função da retirada da ftc. PH3: st_pinza_1_ftc_fermata_polmone_3.
AND HR_213  ; Trida_Sempre Off_010323.
ORLD
ANDLD
SET HR_50105  ; filtro_su_ftc_per_reset_traslazione_quadrotta
LD TR0
AND OUT_10204  ; KM4: polmone 4.
ANDNOT W_112  ; PH4: st_pinza_1_ftc_fermata_polmone_4.
AND W_4003  ; stato_automatico
AND HR_213  ; Trida_Sempre Off_010323.
TIMX(550) 0682 &20  ; Auxiliar em função da retirada da ftc. PH3: st_pinza_1_ftc_fermata_polmone_3.

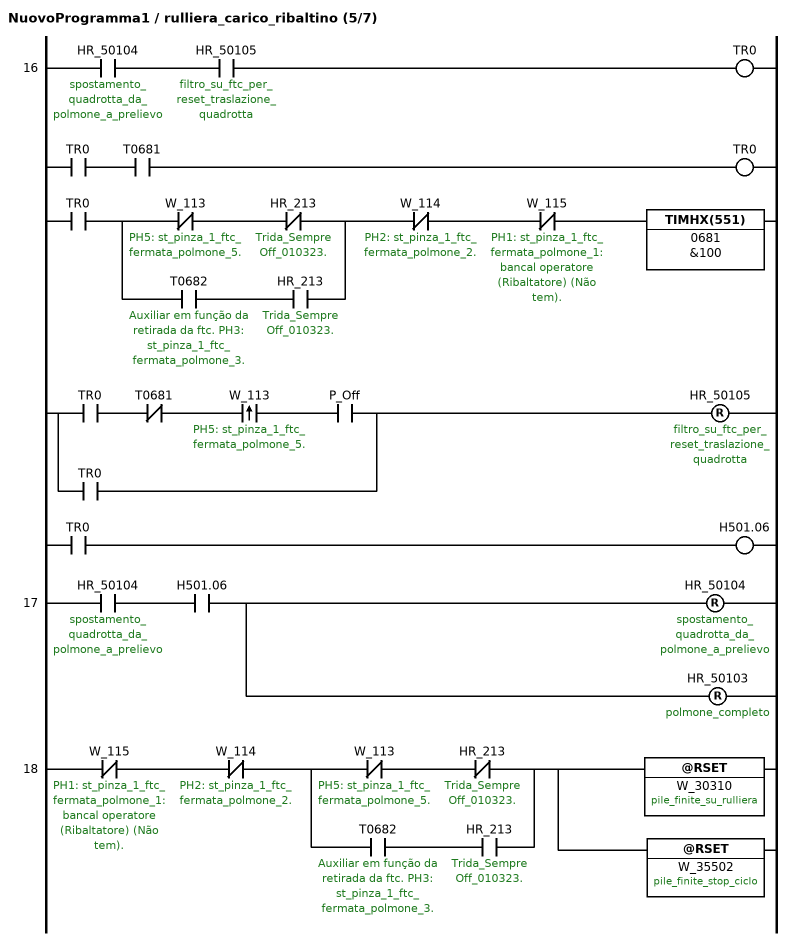
; rung 16
LD HR_50104  ; spostamento_quadrotta_da_polmone_a_prelievo
AND HR_50105  ; filtro_su_ftc_per_reset_traslazione_quadrotta
OUT TR0
LDNOT W_113  ; PH5: st_pinza_1_ftc_fermata_polmone_5.
ANDNOT HR_213  ; Trida_Sempre Off_010323.
LD T0682  ; Auxiliar em função da retirada da ftc. PH3: st_pinza_1_ftc_fermata_polmone_3.
AND HR_213  ; Trida_Sempre Off_010323.
ORLD
ANDLD
ANDNOT W_114  ; PH2: st_pinza_1_ftc_fermata_polmone_2.
ANDNOT W_115  ; PH1: st_pinza_1_ftc_fermata_polmone_1: bancal operatore (Ribaltatore) (Não tem).
TIMHX(551) 0681 &100
LD TR0
ANDNOT T0681
@AND W_113  ; PH5: st_pinza_1_ftc_fermata_polmone_5.
AND P_Off
LD TR0
AND T0681
OUT TR0
ORLD
RSET HR_50105  ; filtro_su_ftc_per_reset_traslazione_quadrotta
LD TR0
OUT H501.06
; rung 17
LD HR_50104  ; spostamento_quadrotta_da_polmone_a_prelievo
AND H501.06
RSET HR_50104  ; spostamento_quadrotta_da_polmone_a_prelievo
RSET HR_50103  ; polmone_completo
; rung 18
LDNOT W_115  ; PH1: st_pinza_1_ftc_fermata_polmone_1: bancal operatore (Ribaltatore) (Não tem).
ANDNOT W_114  ; PH2: st_pinza_1_ftc_fermata_polmone_2.
LDNOT W_113  ; PH5: st_pinza_1_ftc_fermata_polmone_5.
ANDNOT HR_213  ; Trida_Sempre Off_010323.
LD T0682  ; Auxiliar em função da retirada da ftc. PH3: st_pinza_1_ftc_fermata_polmone_3.
AND HR_213  ; Trida_Sempre Off_010323.
ORLD
ANDLD
@RSET W_30310  ; pile_finite_su_rulliera
@RSET W_35502  ; pile_finite_stop_ciclo

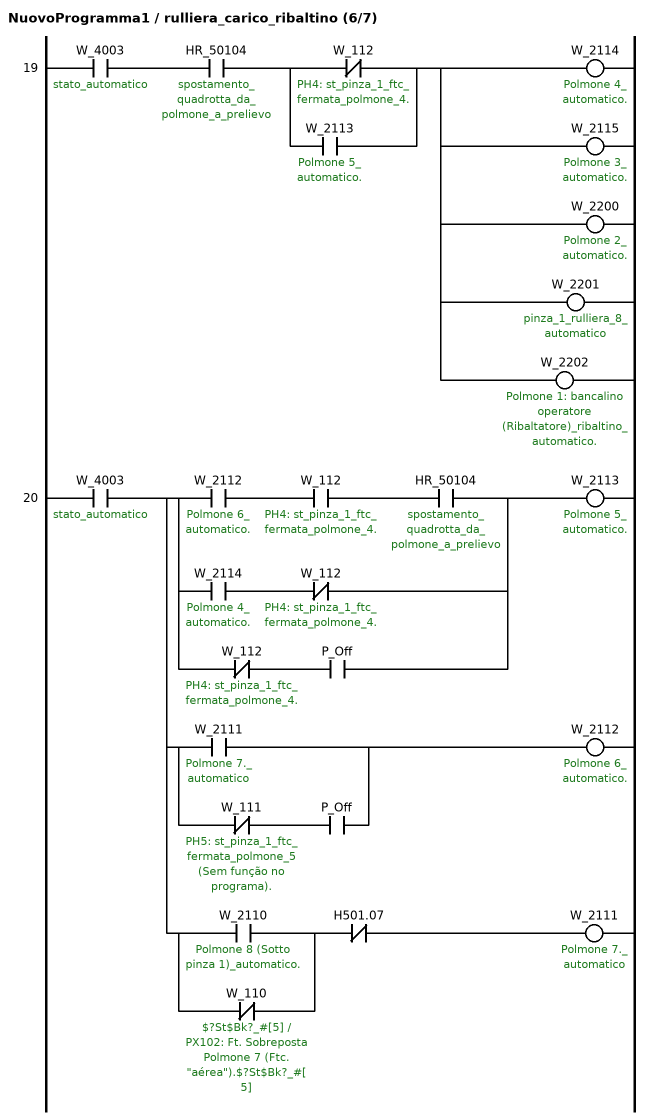
; rung 19
LD W_4003  ; stato_automatico
AND HR_50104  ; spostamento_quadrotta_da_polmone_a_prelievo
LDNOT W_112  ; PH4: st_pinza_1_ftc_fermata_polmone_4.
OR W_2113  ; Polmone 5_automatico.
ANDLD
OUT W_2114  ; Polmone 4_automatico.
OUT W_2115  ; Polmone 3_automatico.
OUT W_2200  ; Polmone 2_automatico.
OUT W_2201  ; pinza_1_rulliera_8_automatico
OUT W_2202  ; Polmone 1: bancalino operatore (Ribaltatore)_ribaltino_automatico.
; rung 20
LD W_4003  ; stato_automatico
OUT TR0
LD W_2112  ; Polmone 6_automatico.
AND W_112  ; PH4: st_pinza_1_ftc_fermata_polmone_4.
AND HR_50104  ; spostamento_quadrotta_da_polmone_a_prelievo
LD W_2114  ; Polmone 4_automatico.
ANDNOT W_112  ; PH4: st_pinza_1_ftc_fermata_polmone_4.
ORLD
LDNOT W_112  ; PH4: st_pinza_1_ftc_fermata_polmone_4.
AND P_Off
ORLD
ANDLD
OUT W_2113  ; Polmone 5_automatico.
LD TR0
LD W_2111  ; Polmone 7._automatico
LDNOT W_111  ; PH5: st_pinza_1_ftc_fermata_polmone_5 (Sem função no programa).
AND P_Off
ORLD
ANDLD
OUT W_2112  ; Polmone 6_automatico.
LD TR0
LD W_2110  ; Polmone 8 (Sotto pinza 1)_automatico.
ORNOT W_110  ; $?St$Bk?_#[5] / PX102: Ft. Sobreposta Polmone 7 (Ftc. "aérea").$?St$Bk?_#[5]
ANDLD
ANDNOT H501.07
OUT W_2111  ; Polmone 7._automatico

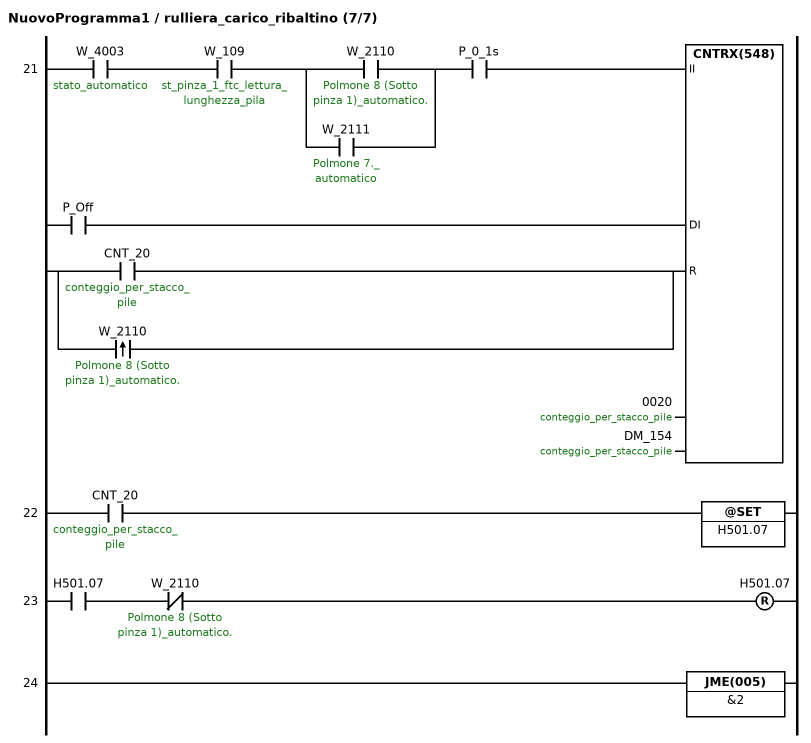
; rung 21
LD W_4003  ; stato_automatico
AND W_109  ; st_pinza_1_ftc_lettura_lunghezza_pila
LD W_2110  ; Polmone 8 (Sotto pinza 1)_automatico.
OR W_2111  ; Polmone 7._automatico
ANDLD
AND P_0_1s
LD P_Off
LD CNT_20  ; conteggio_per_stacco_pile
@OR W_2110  ; Polmone 8 (Sotto pinza 1)_automatico.
CNTRX(548) 0020 DM_154  ; conteggio_per_stacco_pile
; rung 22
LD CNT_20  ; conteggio_per_stacco_pile
@SET H501.07
; rung 23
LD H501.07
ANDNOT W_2110  ; Polmone 8 (Sotto pinza 1)_automatico.
RSET H501.07
; rung 24
JME(005) &2

### Section automatico_pinza_pallet

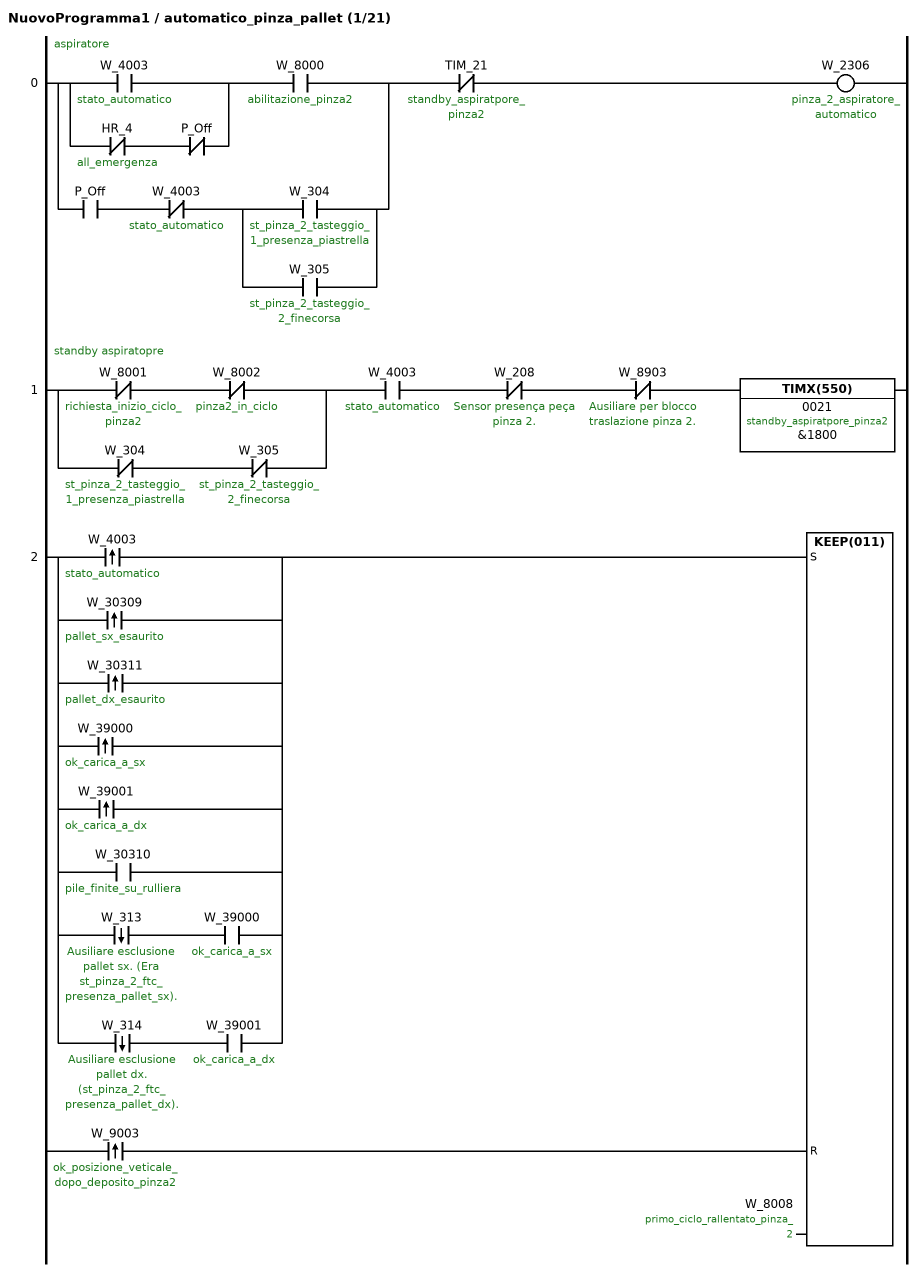
; rung 0: aspiratore
LD W_4003  ; stato_automatico
LDNOT HR_4  ; all_emergenza
ANDNOT P_Off
ORLD
AND W_8000  ; abilitazione_pinza2
LD P_Off
ANDNOT W_4003  ; stato_automatico
LD W_304  ; st_pinza_2_tasteggio_1_presenza_piastrella
OR W_305  ; st_pinza_2_tasteggio_2_finecorsa
ANDLD
ORLD
ANDNOT TIM_21  ; standby_aspiratpore_pinza2
OUT W_2306  ; pinza_2_aspiratore_automatico
; rung 1: standby aspiratopre
LDNOT W_8001  ; richiesta_inizio_ciclo_pinza2
ANDNOT W_8002  ; pinza2_in_ciclo
LDNOT W_304  ; st_pinza_2_tasteggio_1_presenza_piastrella
ANDNOT W_305  ; st_pinza_2_tasteggio_2_finecorsa
ORLD
AND W_4003  ; stato_automatico
ANDNOT W_208  ; Sensor presença peça pinza 2.
ANDNOT W_8903  ; Ausiliare per blocco traslazione pinza 2.
TIMX(550) 0021 &1800  ; standby_aspiratpore_pinza2
; rung 2
@LD W_4003  ; stato_automatico
@OR W_30309  ; pallet_sx_esaurito
@OR W_30311  ; pallet_dx_esaurito
@OR W_39000  ; ok_carica_a_sx
@OR W_39001  ; ok_carica_a_dx
OR W_30310  ; pile_finite_su_rulliera
%LD W_313  ; Ausiliare esclusione pallet sx. (Era st_pinza_2_ftc_presenza_pallet_sx).
AND W_39000  ; ok_carica_a_sx
ORLD
%LD W_314  ; Ausiliare esclusione pallet dx. (st_pinza_2_ftc_presenza_pallet_dx).
AND W_39001  ; ok_carica_a_dx
ORLD
@LD W_9003  ; ok_posizione_veticale_dopo_deposito_pinza2
KEEP(011) W_8008  ; primo_ciclo_rallentato_pinza_2

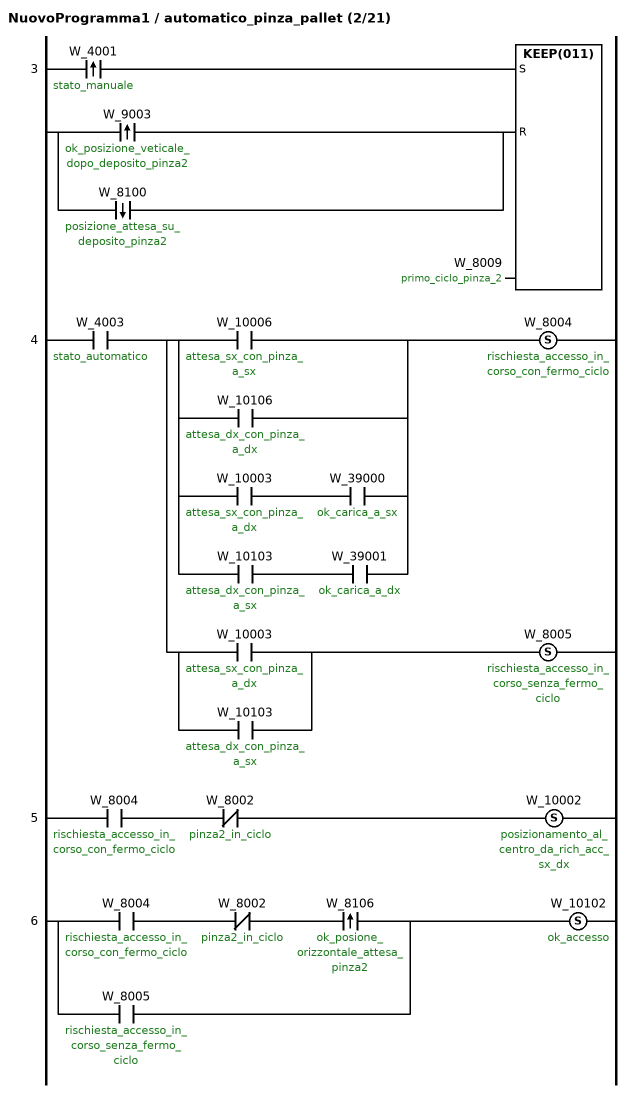
; rung 3
@LD W_4001  ; stato_manuale
@LD W_9003  ; ok_posizione_veticale_dopo_deposito_pinza2
%OR W_8100  ; posizione_attesa_su_deposito_pinza2
KEEP(011) W_8009  ; primo_ciclo_pinza_2
; rung 4
LD W_4003  ; stato_automatico
OUT TR0
LD W_10006  ; attesa_sx_con_pinza_a_sx
OR W_10106  ; attesa_dx_con_pinza_a_dx
LD W_10003  ; attesa_sx_con_pinza_a_dx
AND W_39000  ; ok_carica_a_sx
ORLD
LD W_10103  ; attesa_dx_con_pinza_a_sx
AND W_39001  ; ok_carica_a_dx
ORLD
ANDLD
SET W_8004  ; rischiesta_accesso_in_corso_con_fermo_ciclo
LD TR0
LD W_10003  ; attesa_sx_con_pinza_a_dx
OR W_10103  ; attesa_dx_con_pinza_a_sx
ANDLD
SET W_8005  ; rischiesta_accesso_in_corso_senza_fermo_ciclo
; rung 5
LD W_8004  ; rischiesta_accesso_in_corso_con_fermo_ciclo
ANDNOT W_8002  ; pinza2_in_ciclo
SET W_10002  ; posizionamento_al_centro_da_rich_acc_sx_dx
; rung 6
LD W_8004  ; rischiesta_accesso_in_corso_con_fermo_ciclo
ANDNOT W_8002  ; pinza2_in_ciclo
@AND W_8106  ; ok_posione_orizzontale_attesa_pinza2
OR W_8005  ; rischiesta_accesso_in_corso_senza_fermo_ciclo
SET W_10102  ; ok_accesso

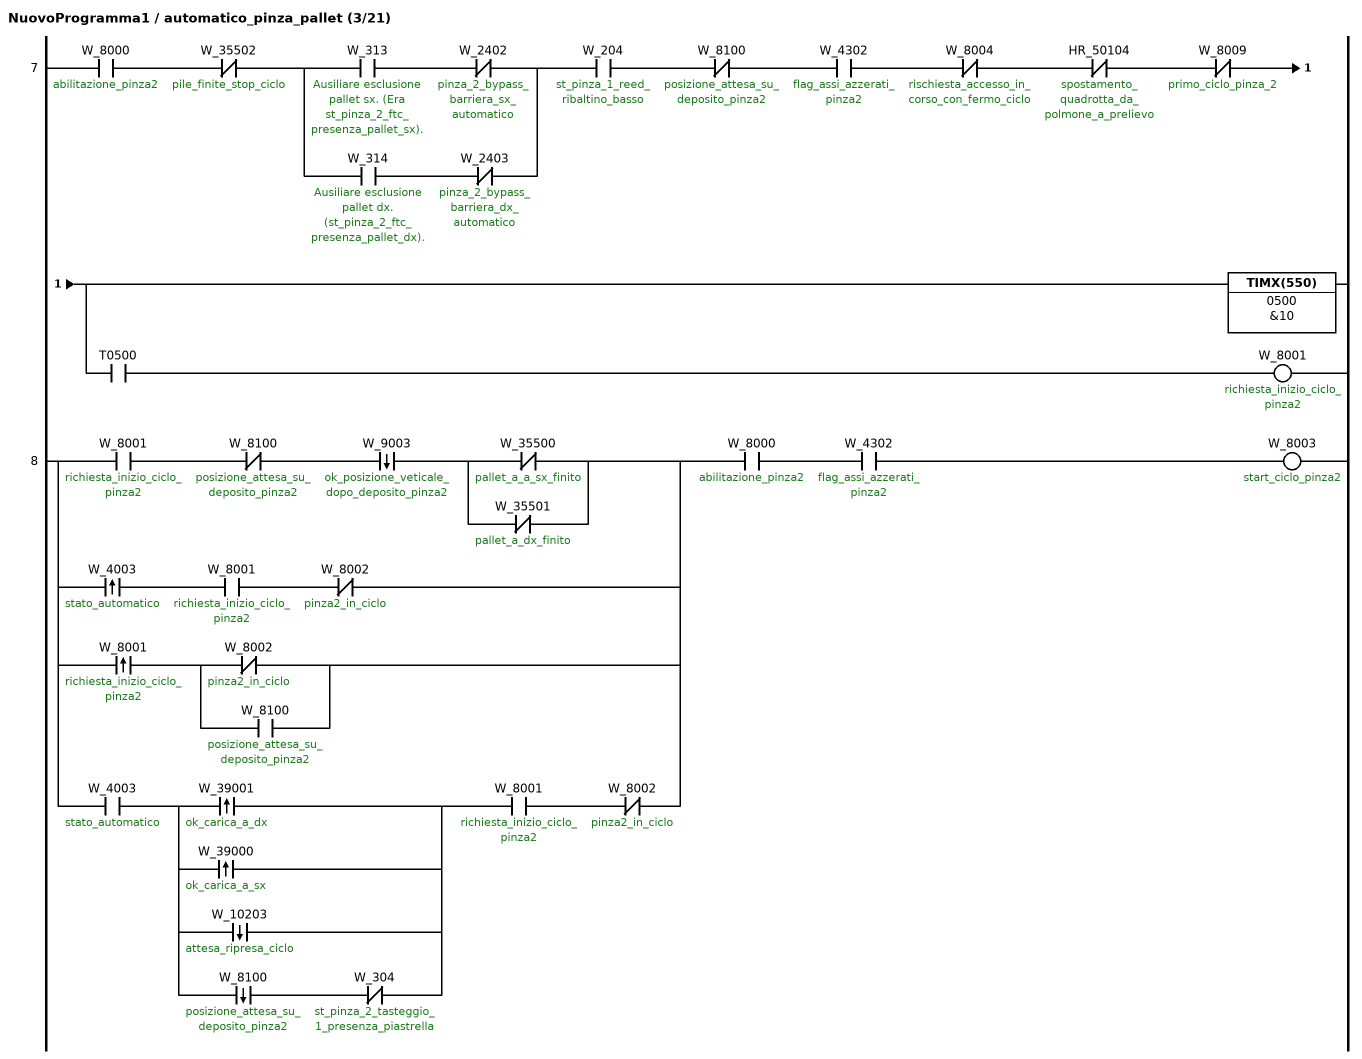
; rung 7
LD W_8000  ; abilitazione_pinza2
ANDNOT W_35502  ; pile_finite_stop_ciclo
LD W_313  ; Ausiliare esclusione pallet sx. (Era st_pinza_2_ftc_presenza_pallet_sx).
ANDNOT W_2402  ; pinza_2_bypass_barriera_sx_automatico
LD W_314  ; Ausiliare esclusione pallet dx. (st_pinza_2_ftc_presenza_pallet_dx).
ANDNOT W_2403  ; pinza_2_bypass_barriera_dx_automatico
ORLD
ANDLD
AND W_204  ; st_pinza_1_reed_ribaltino_basso
ANDNOT W_8100  ; posizione_attesa_su_deposito_pinza2
AND W_4302  ; flag_assi_azzerati_pinza2
ANDNOT W_8004  ; rischiesta_accesso_in_corso_con_fermo_ciclo
ANDNOT HR_50104  ; spostamento_quadrotta_da_polmone_a_prelievo
ANDNOT W_8009  ; primo_ciclo_pinza_2
TIMX(550) 0500 &10
AND T0500
OUT W_8001  ; richiesta_inizio_ciclo_pinza2
; rung 8
LD W_8001  ; richiesta_inizio_ciclo_pinza2
ANDNOT W_8100  ; posizione_attesa_su_deposito_pinza2
%AND W_9003  ; ok_posizione_veticale_dopo_deposito_pinza2
LDNOT W_35500  ; pallet_a_a_sx_finito
ORNOT W_35501  ; pallet_a_dx_finito
ANDLD
@LD W_4003  ; stato_automatico
AND W_8001  ; richiesta_inizio_ciclo_pinza2
ANDNOT W_8002  ; pinza2_in_ciclo
ORLD
@LD W_8001  ; richiesta_inizio_ciclo_pinza2
LDNOT W_8002  ; pinza2_in_ciclo
OR W_8100  ; posizione_attesa_su_deposito_pinza2
ANDLD
ORLD
LD W_4003  ; stato_automatico
@LD W_39001  ; ok_carica_a_dx
@OR W_39000  ; ok_carica_a_sx
%OR W_10203  ; attesa_ripresa_ciclo
%LD W_8100  ; posizione_attesa_su_deposito_pinza2
ANDNOT W_304  ; st_pinza_2_tasteggio_1_presenza_piastrella
ORLD
ANDLD
AND W_8001  ; richiesta_inizio_ciclo_pinza2
ANDNOT W_8002  ; pinza2_in_ciclo
ORLD
AND W_8000  ; abilitazione_pinza2
AND W_4302  ; flag_assi_azzerati_pinza2
OUT W_8003  ; start_ciclo_pinza2

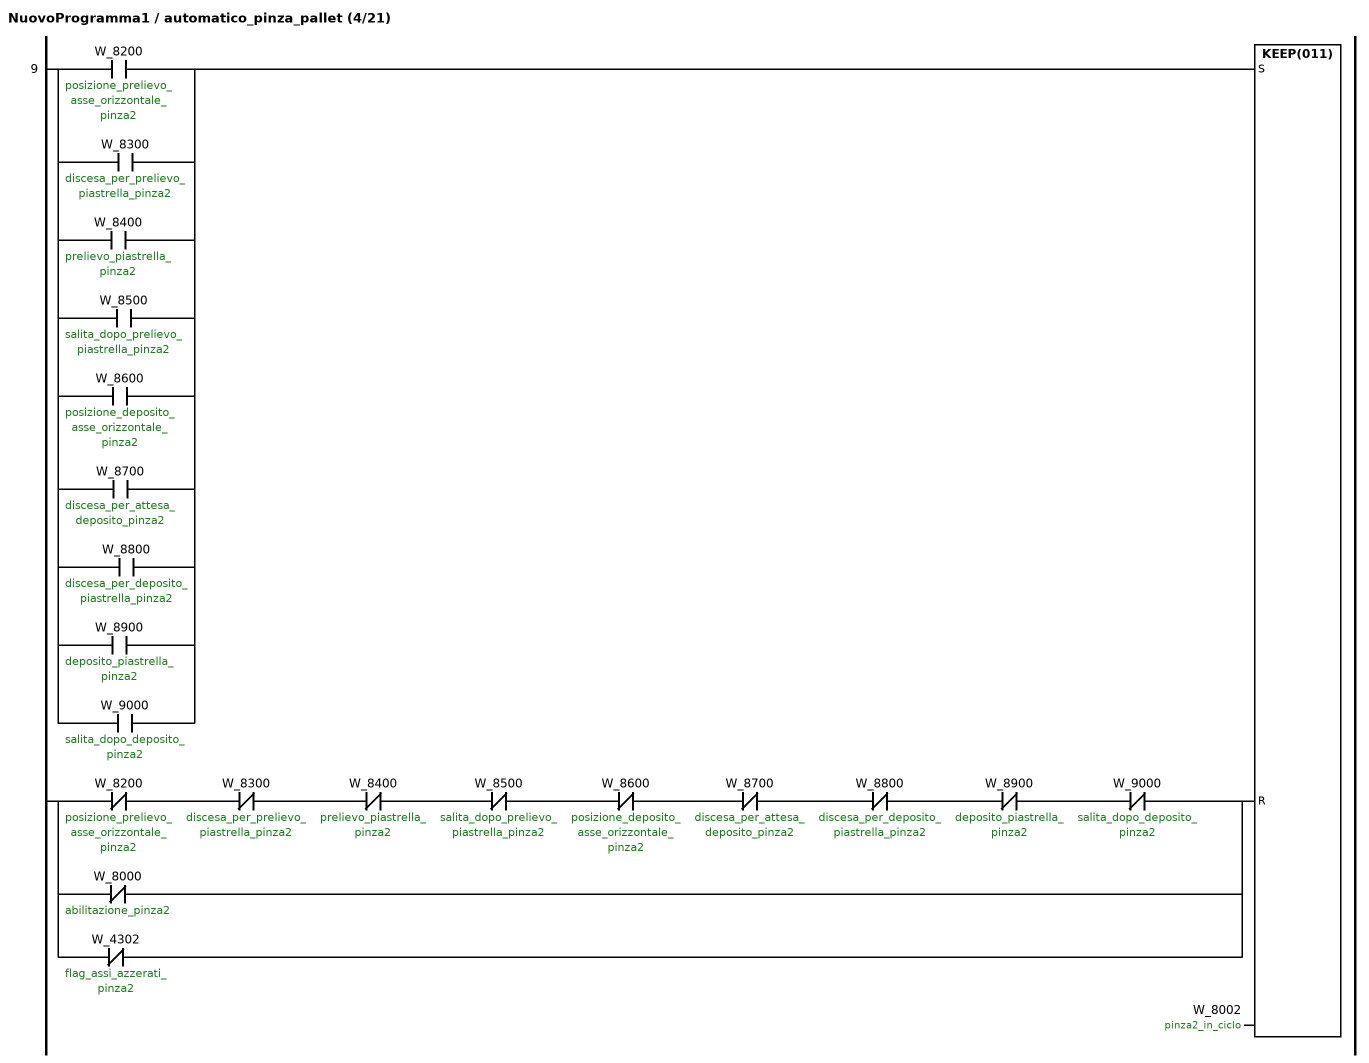
; rung 9
LD W_8200  ; posizione_prelievo_asse_orizzontale_pinza2
OR W_8300  ; discesa_per_prelievo_piastrella_pinza2
OR W_8400  ; prelievo_piastrella_pinza2
OR W_8500  ; salita_dopo_prelievo_piastrella_pinza2
OR W_8600  ; posizione_deposito_asse_orizzontale_pinza2
OR W_8700  ; discesa_per_attesa_deposito_pinza2
OR W_8800  ; discesa_per_deposito_piastrella_pinza2
OR W_8900  ; deposito_piastrella_pinza2
OR W_9000  ; salita_dopo_deposito_pinza2
LDNOT W_8200  ; posizione_prelievo_asse_orizzontale_pinza2
ANDNOT W_8300  ; discesa_per_prelievo_piastrella_pinza2
ANDNOT W_8400  ; prelievo_piastrella_pinza2
ANDNOT W_8500  ; salita_dopo_prelievo_piastrella_pinza2
ANDNOT W_8600  ; posizione_deposito_asse_orizzontale_pinza2
ANDNOT W_8700  ; discesa_per_attesa_deposito_pinza2
ANDNOT W_8800  ; discesa_per_deposito_piastrella_pinza2
ANDNOT W_8900  ; deposito_piastrella_pinza2
ANDNOT W_9000  ; salita_dopo_deposito_pinza2
ORNOT W_8000  ; abilitazione_pinza2
ORNOT W_4302  ; flag_assi_azzerati_pinza2
KEEP(011) W_8002  ; pinza2_in_ciclo

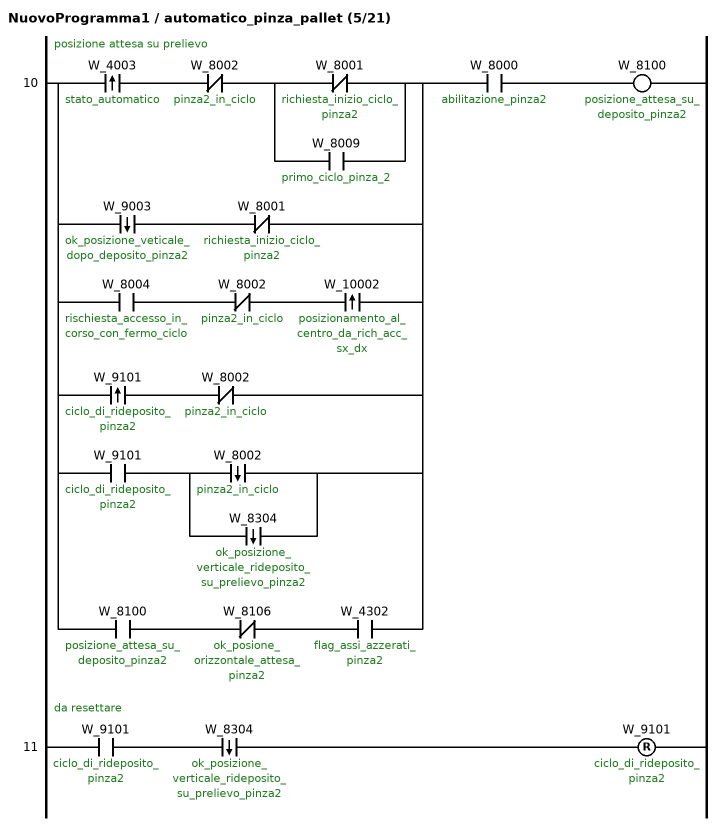
; rung 10: posizione attesa su prelievo
@LD W_4003  ; stato_automatico
ANDNOT W_8002  ; pinza2_in_ciclo
LDNOT W_8001  ; richiesta_inizio_ciclo_pinza2
OR W_8009  ; primo_ciclo_pinza_2
ANDLD
%LD W_9003  ; ok_posizione_veticale_dopo_deposito_pinza2
ANDNOT W_8001  ; richiesta_inizio_ciclo_pinza2
ORLD
LD W_8004  ; rischiesta_accesso_in_corso_con_fermo_ciclo
ANDNOT W_8002  ; pinza2_in_ciclo
@AND W_10002  ; posizionamento_al_centro_da_rich_acc_sx_dx
ORLD
@LD W_9101  ; ciclo_di_rideposito_pinza2
ANDNOT W_8002  ; pinza2_in_ciclo
ORLD
LD W_9101  ; ciclo_di_rideposito_pinza2
%LD W_8002  ; pinza2_in_ciclo
%OR W_8304  ; ok_posizione_verticale_rideposito_su_prelievo_pinza2
ANDLD
ORLD
LD W_8100  ; posizione_attesa_su_deposito_pinza2
ANDNOT W_8106  ; ok_posione_orizzontale_attesa_pinza2
AND W_4302  ; flag_assi_azzerati_pinza2
ORLD
AND W_8000  ; abilitazione_pinza2
OUT W_8100  ; posizione_attesa_su_deposito_pinza2
; rung 11: da resettare
LD W_9101  ; ciclo_di_rideposito_pinza2
%AND W_8304  ; ok_posizione_verticale_rideposito_su_prelievo_pinza2
RSET W_9101  ; ciclo_di_rideposito_pinza2

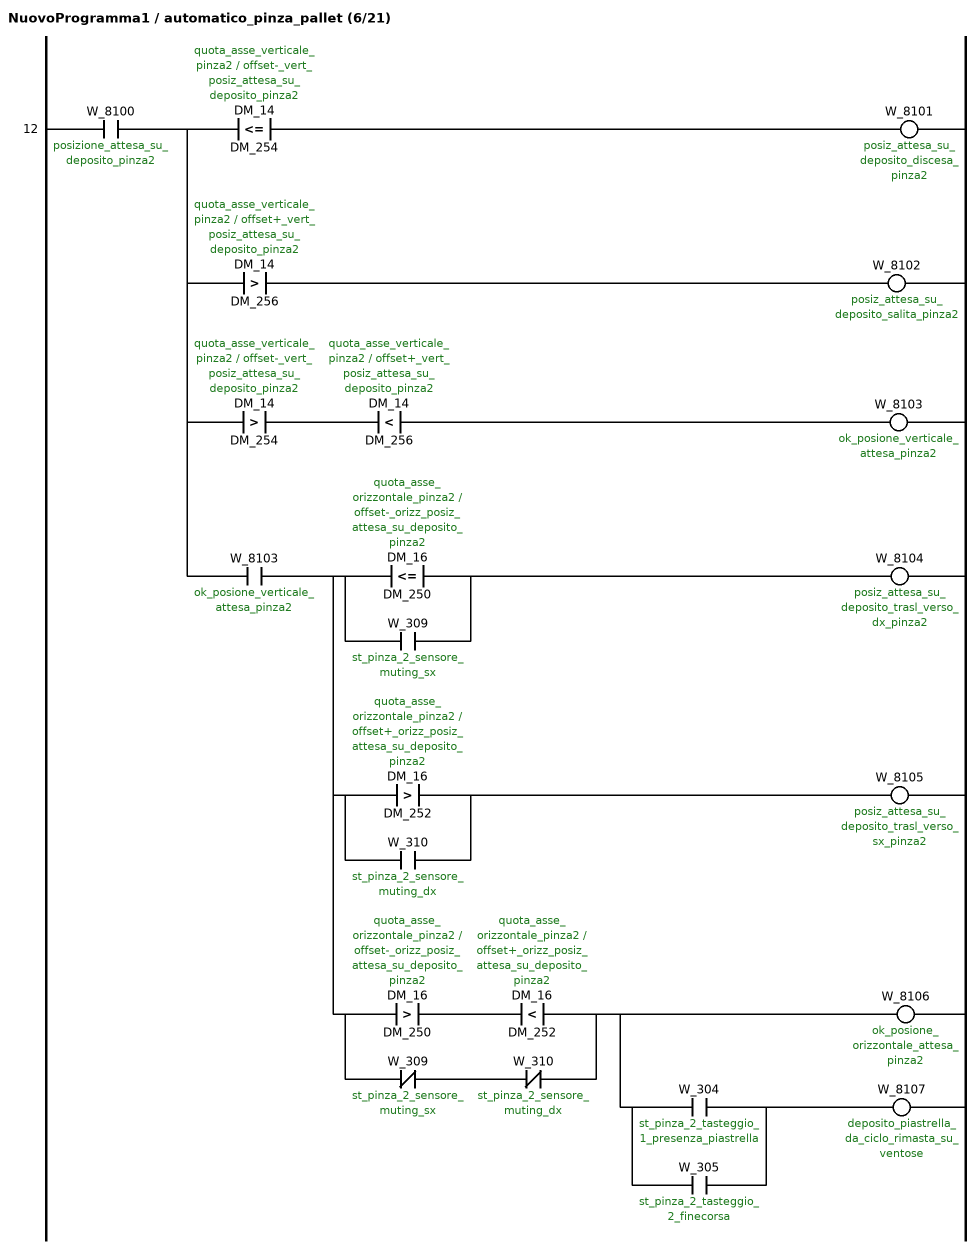
; rung 12
LD W_8100  ; posizione_attesa_su_deposito_pinza2
OUT TR0
AND<=SL(318) DM_14 DM_254  ; quota_asse_verticale_pinza2, offset-_vert_posiz_attesa_su_deposito_pinza2
OUT W_8101  ; posiz_attesa_su_deposito_discesa_pinza2
LD TR0
AND>SL(323) DM_14 DM_256  ; quota_asse_verticale_pinza2, offset+_vert_posiz_attesa_su_deposito_pinza2
OUT W_8102  ; posiz_attesa_su_deposito_salita_pinza2
LD TR0
AND>SL(323) DM_14 DM_254  ; quota_asse_verticale_pinza2, offset-_vert_posiz_attesa_su_deposito_pinza2
AND<SL(313) DM_14 DM_256  ; quota_asse_verticale_pinza2, offset+_vert_posiz_attesa_su_deposito_pinza2
OUT W_8103  ; ok_posione_verticale_attesa_pinza2
LD TR0
AND W_8103  ; ok_posione_verticale_attesa_pinza2
OUT TR0
LD<=SL(318) DM_16 DM_250  ; quota_asse_orizzontale_pinza2, offset-_orizz_posiz_attesa_su_deposito_pinza2
OR W_309  ; st_pinza_2_sensore_muting_sx
ANDLD
OUT W_8104  ; posiz_attesa_su_deposito_trasl_verso_dx_pinza2
LD TR0
LD>SL(323) DM_16 DM_252  ; quota_asse_orizzontale_pinza2, offset+_orizz_posiz_attesa_su_deposito_pinza2
OR W_310  ; st_pinza_2_sensore_muting_dx
ANDLD
OUT W_8105  ; posiz_attesa_su_deposito_trasl_verso_sx_pinza2
LD TR0
LD>SL(323) DM_16 DM_250  ; quota_asse_orizzontale_pinza2, offset-_orizz_posiz_attesa_su_deposito_pinza2
AND<SL(313) DM_16 DM_252  ; quota_asse_orizzontale_pinza2, offset+_orizz_posiz_attesa_su_deposito_pinza2
LDNOT W_309  ; st_pinza_2_sensore_muting_sx
ANDNOT W_310  ; st_pinza_2_sensore_muting_dx
ORLD
ANDLD
OUT W_8106  ; ok_posione_orizzontale_attesa_pinza2
LD W_304  ; st_pinza_2_tasteggio_1_presenza_piastrella
OR W_305  ; st_pinza_2_tasteggio_2_finecorsa
ANDLD
OUT W_8107  ; deposito_piastrella_da_ciclo_rimasta_su_ventose

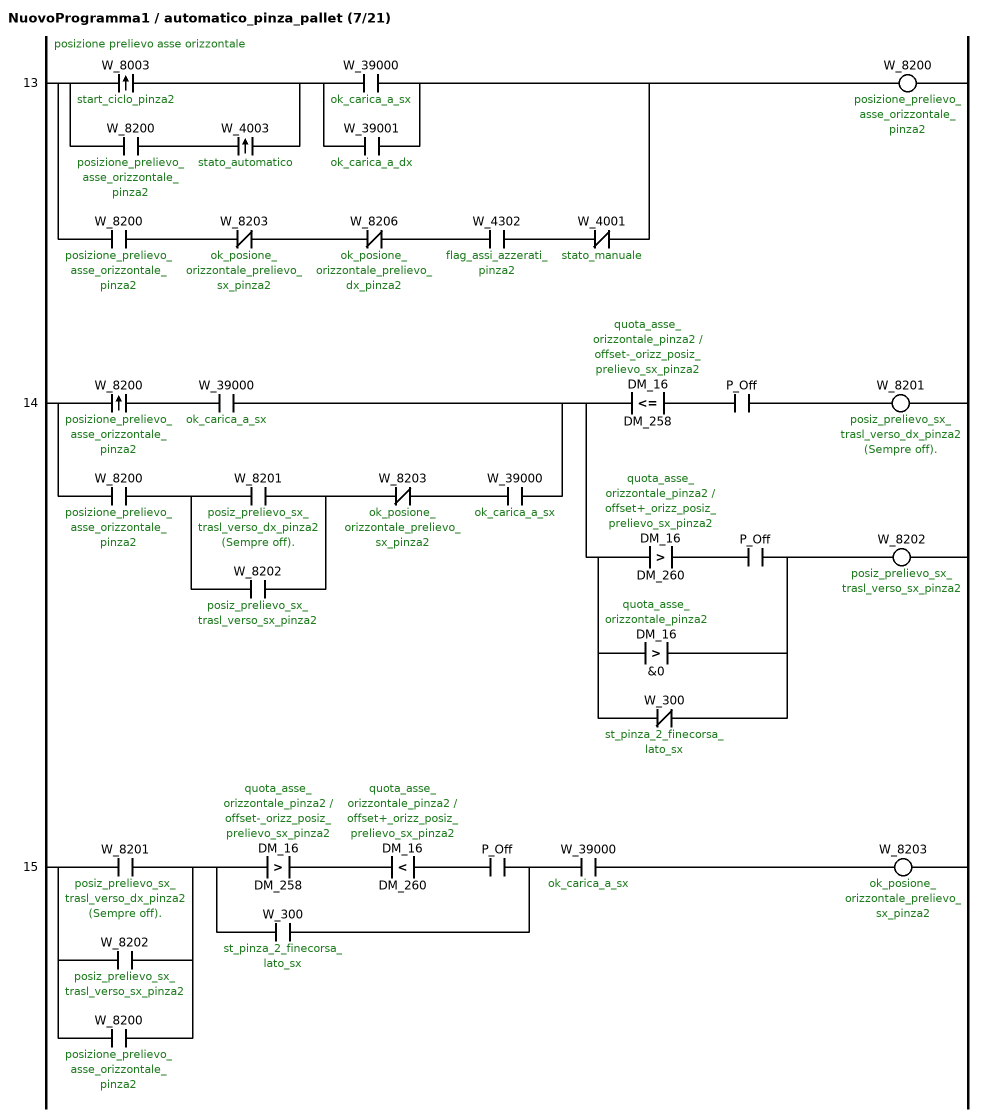
; rung 13: posizione prelievo asse orizzontale
@LD W_8003  ; start_ciclo_pinza2
LD W_8200  ; posizione_prelievo_asse_orizzontale_pinza2
@AND W_4003  ; stato_automatico
ORLD
LD W_39000  ; ok_carica_a_sx
OR W_39001  ; ok_carica_a_dx
ANDLD
LD W_8200  ; posizione_prelievo_asse_orizzontale_pinza2
ANDNOT W_8203  ; ok_posione_orizzontale_prelievo_sx_pinza2
ANDNOT W_8206  ; ok_posione_orizzontale_prelievo_dx_pinza2
AND W_4302  ; flag_assi_azzerati_pinza2
ANDNOT W_4001  ; stato_manuale
ORLD
OUT W_8200  ; posizione_prelievo_asse_orizzontale_pinza2
; rung 14
@LD W_8200  ; posizione_prelievo_asse_orizzontale_pinza2
AND W_39000  ; ok_carica_a_sx
LD W_8200  ; posizione_prelievo_asse_orizzontale_pinza2
LD W_8201  ; posiz_prelievo_sx_trasl_verso_dx_pinza2 (Sempre off).
OR W_8202  ; posiz_prelievo_sx_trasl_verso_sx_pinza2
ANDLD
ANDNOT W_8203  ; ok_posione_orizzontale_prelievo_sx_pinza2
AND W_39000  ; ok_carica_a_sx
ORLD
OUT TR0
AND<=SL(318) DM_16 DM_258  ; quota_asse_orizzontale_pinza2, offset-_orizz_posiz_prelievo_sx_pinza2
AND P_Off
OUT W_8201  ; posiz_prelievo_sx_trasl_verso_dx_pinza2 (Sempre off).
LD TR0
LD>SL(323) DM_16 DM_260  ; quota_asse_orizzontale_pinza2, offset+_orizz_posiz_prelievo_sx_pinza2
AND P_Off
OR>SL(323) DM_16 &0  ; quota_asse_orizzontale_pinza2
ORNOT W_300  ; st_pinza_2_finecorsa_lato_sx
ANDLD
OUT W_8202  ; posiz_prelievo_sx_trasl_verso_sx_pinza2
; rung 15
LD W_8201  ; posiz_prelievo_sx_trasl_verso_dx_pinza2 (Sempre off).
OR W_8202  ; posiz_prelievo_sx_trasl_verso_sx_pinza2
OR W_8200  ; posizione_prelievo_asse_orizzontale_pinza2
LD>SL(323) DM_16 DM_258  ; quota_asse_orizzontale_pinza2, offset-_orizz_posiz_prelievo_sx_pinza2
AND<SL(313) DM_16 DM_260  ; quota_asse_orizzontale_pinza2, offset+_orizz_posiz_prelievo_sx_pinza2
AND P_Off
OR W_300  ; st_pinza_2_finecorsa_lato_sx
ANDLD
AND W_39000  ; ok_carica_a_sx
OUT W_8203  ; ok_posione_orizzontale_prelievo_sx_pinza2

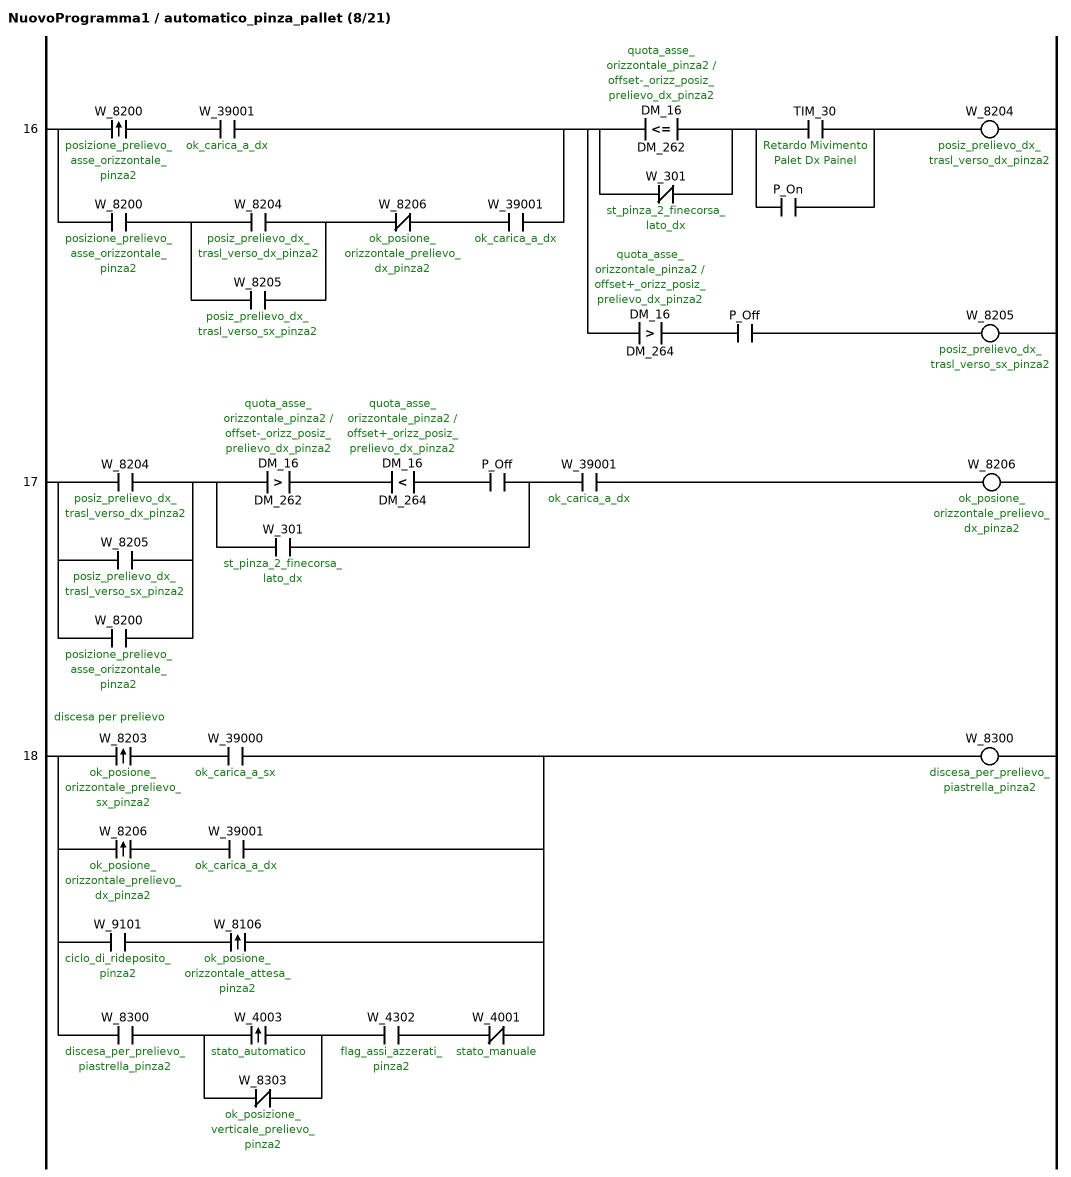
; rung 16
@LD W_8200  ; posizione_prelievo_asse_orizzontale_pinza2
AND W_39001  ; ok_carica_a_dx
LD W_8200  ; posizione_prelievo_asse_orizzontale_pinza2
LD W_8204  ; posiz_prelievo_dx_trasl_verso_dx_pinza2
OR W_8205  ; posiz_prelievo_dx_trasl_verso_sx_pinza2
ANDLD
ANDNOT W_8206  ; ok_posione_orizzontale_prelievo_dx_pinza2
AND W_39001  ; ok_carica_a_dx
ORLD
OUT TR0
LD<=SL(318) DM_16 DM_262  ; quota_asse_orizzontale_pinza2, offset-_orizz_posiz_prelievo_dx_pinza2
ORNOT W_301  ; st_pinza_2_finecorsa_lato_dx
ANDLD
LD TIM_30  ; Retardo Mivimento Palet Dx Painel
OR P_On
ANDLD
OUT W_8204  ; posiz_prelievo_dx_trasl_verso_dx_pinza2
LD TR0
AND>SL(323) DM_16 DM_264  ; quota_asse_orizzontale_pinza2, offset+_orizz_posiz_prelievo_dx_pinza2
AND P_Off
OUT W_8205  ; posiz_prelievo_dx_trasl_verso_sx_pinza2
; rung 17
LD W_8204  ; posiz_prelievo_dx_trasl_verso_dx_pinza2
OR W_8205  ; posiz_prelievo_dx_trasl_verso_sx_pinza2
OR W_8200  ; posizione_prelievo_asse_orizzontale_pinza2
LD>SL(323) DM_16 DM_262  ; quota_asse_orizzontale_pinza2, offset-_orizz_posiz_prelievo_dx_pinza2
AND<SL(313) DM_16 DM_264  ; quota_asse_orizzontale_pinza2, offset+_orizz_posiz_prelievo_dx_pinza2
AND P_Off
OR W_301  ; st_pinza_2_finecorsa_lato_dx
ANDLD
AND W_39001  ; ok_carica_a_dx
OUT W_8206  ; ok_posione_orizzontale_prelievo_dx_pinza2
; rung 18: discesa per prelievo
@LD W_8203  ; ok_posione_orizzontale_prelievo_sx_pinza2
AND W_39000  ; ok_carica_a_sx
@LD W_8206  ; ok_posione_orizzontale_prelievo_dx_pinza2
AND W_39001  ; ok_carica_a_dx
ORLD
LD W_9101  ; ciclo_di_rideposito_pinza2
@AND W_8106  ; ok_posione_orizzontale_attesa_pinza2
ORLD
LD W_8300  ; discesa_per_prelievo_piastrella_pinza2
@LD W_4003  ; stato_automatico
ORNOT W_8303  ; ok_posizione_verticale_prelievo_pinza2
ANDLD
AND W_4302  ; flag_assi_azzerati_pinza2
ANDNOT W_4001  ; stato_manuale
ORLD
OUT W_8300  ; discesa_per_prelievo_piastrella_pinza2

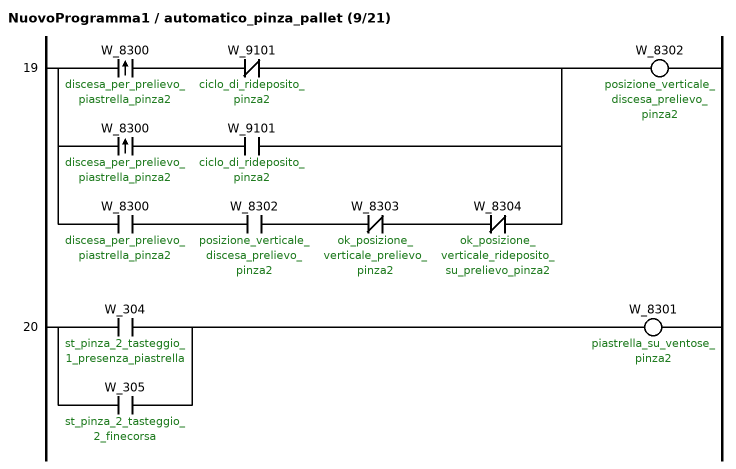
; rung 19
@LD W_8300  ; discesa_per_prelievo_piastrella_pinza2
ANDNOT W_9101  ; ciclo_di_rideposito_pinza2
@LD W_8300  ; discesa_per_prelievo_piastrella_pinza2
AND W_9101  ; ciclo_di_rideposito_pinza2
ORLD
LD W_8300  ; discesa_per_prelievo_piastrella_pinza2
AND W_8302  ; posizione_verticale_discesa_prelievo_pinza2
ANDNOT W_8303  ; ok_posizione_verticale_prelievo_pinza2
ANDNOT W_8304  ; ok_posizione_verticale_rideposito_su_prelievo_pinza2
ORLD
OUT W_8302  ; posizione_verticale_discesa_prelievo_pinza2
; rung 20
LD W_304  ; st_pinza_2_tasteggio_1_presenza_piastrella
OR W_305  ; st_pinza_2_tasteggio_2_finecorsa
OUT W_8301  ; piastrella_su_ventose_pinza2

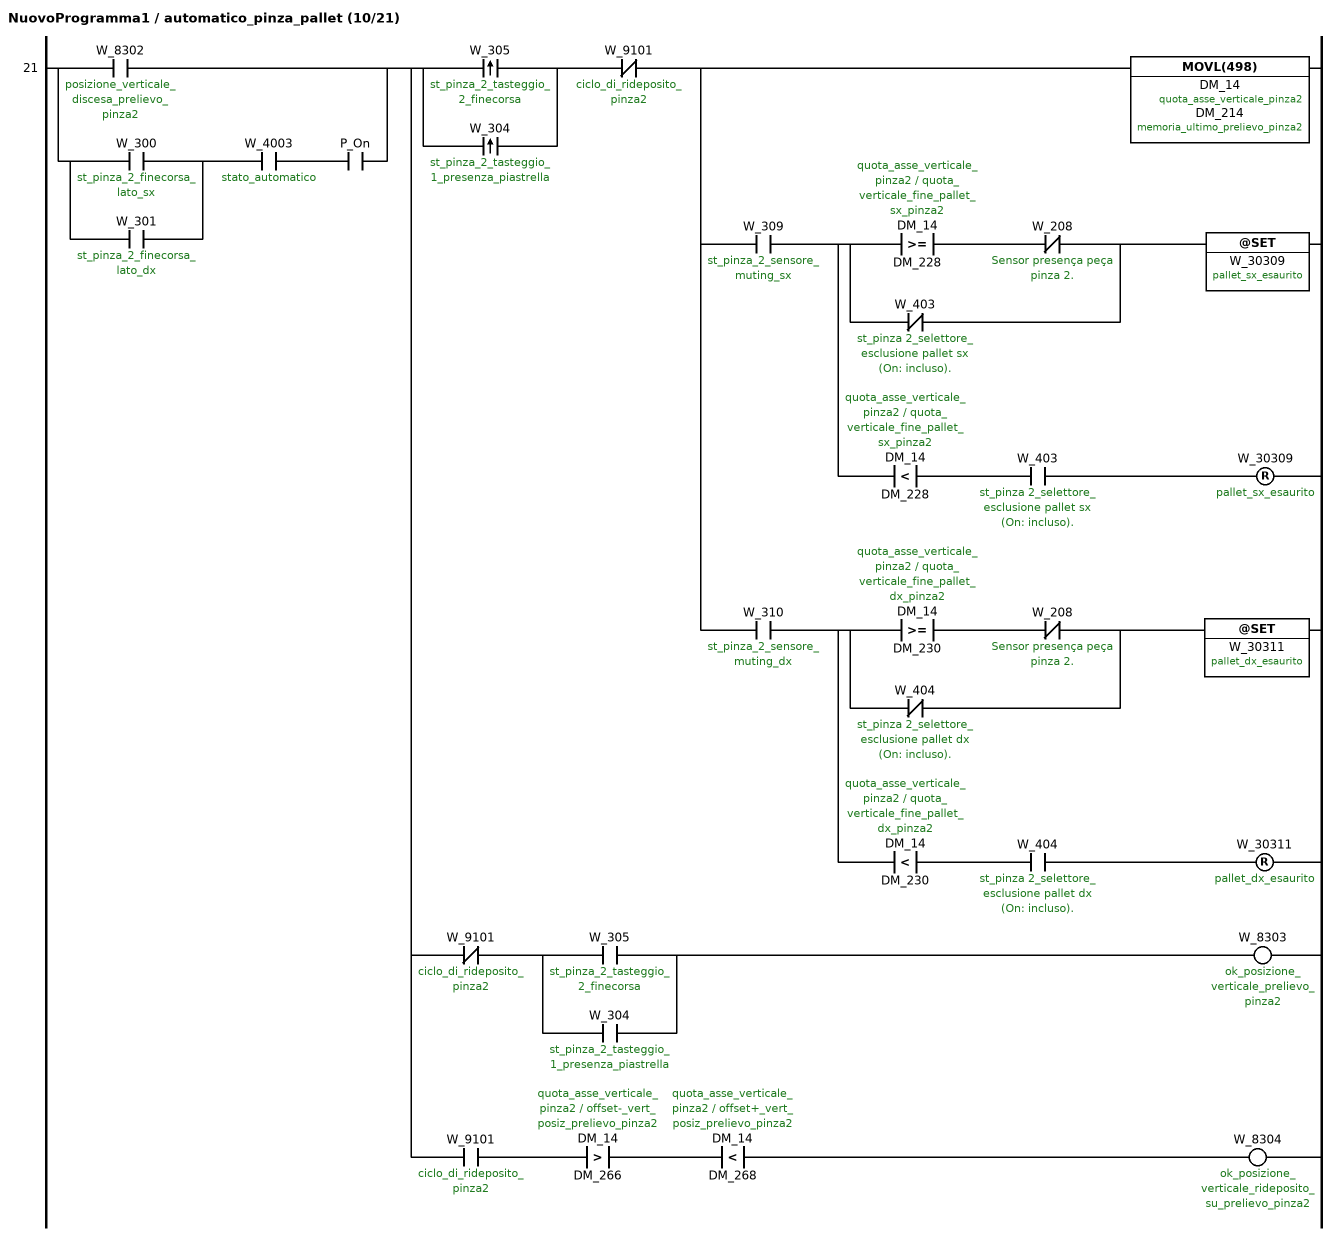
; rung 21
LD W_8302  ; posizione_verticale_discesa_prelievo_pinza2
LD W_300  ; st_pinza_2_finecorsa_lato_sx
OR W_301  ; st_pinza_2_finecorsa_lato_dx
AND W_4003  ; stato_automatico
AND P_On
ORLD
OUT TR0
@LD W_305  ; st_pinza_2_tasteggio_2_finecorsa
@OR W_304  ; st_pinza_2_tasteggio_1_presenza_piastrella
ANDLD
ANDNOT W_9101  ; ciclo_di_rideposito_pinza2
OUT TR1
MOVL(498) DM_14 DM_214  ; quota_asse_verticale_pinza2, memoria_ultimo_prelievo_pinza2
AND W_309  ; st_pinza_2_sensore_muting_sx
OUT TR2
LD>=SL(328) DM_14 DM_228  ; quota_asse_verticale_pinza2, quota_verticale_fine_pallet_sx_pinza2
ANDNOT W_208  ; Sensor presença peça pinza 2.
ORNOT W_403  ; st_pinza 2_selettore_esclusione pallet sx (On: incluso).
ANDLD
@SET W_30309  ; pallet_sx_esaurito
LD TR2
AND<SL(313) DM_14 DM_228  ; quota_asse_verticale_pinza2, quota_verticale_fine_pallet_sx_pinza2
AND W_403  ; st_pinza 2_selettore_esclusione pallet sx (On: incluso).
RSET W_30309  ; pallet_sx_esaurito
LD TR1
AND W_310  ; st_pinza_2_sensore_muting_dx
OUT TR1
LD>=SL(328) DM_14 DM_230  ; quota_asse_verticale_pinza2, quota_verticale_fine_pallet_dx_pinza2
ANDNOT W_208  ; Sensor presença peça pinza 2.
ORNOT W_404  ; st_pinza 2_selettore_esclusione pallet dx (On: incluso).
ANDLD
@SET W_30311  ; pallet_dx_esaurito
LD TR1
AND<SL(313) DM_14 DM_230  ; quota_asse_verticale_pinza2, quota_verticale_fine_pallet_dx_pinza2
AND W_404  ; st_pinza 2_selettore_esclusione pallet dx (On: incluso).
RSET W_30311  ; pallet_dx_esaurito
LD TR0
ANDNOT W_9101  ; ciclo_di_rideposito_pinza2
LD W_305  ; st_pinza_2_tasteggio_2_finecorsa
OR W_304  ; st_pinza_2_tasteggio_1_presenza_piastrella
ANDLD
OUT W_8303  ; ok_posizione_verticale_prelievo_pinza2
LD TR0
AND W_9101  ; ciclo_di_rideposito_pinza2
AND>SL(323) DM_14 DM_266  ; quota_asse_verticale_pinza2, offset-_vert_posiz_prelievo_pinza2
AND<SL(313) DM_14 DM_268  ; quota_asse_verticale_pinza2, offset+_vert_posiz_prelievo_pinza2
OUT W_8304  ; ok_posizione_verticale_rideposito_su_prelievo_pinza2

